LIN {X 0,Y 192.338,Z 600.856,A -85,B 0,C 180,E1 -21672.999,E2 -21672.999} C_VEL
LIN {X 0,Y 190.84,Z 603.624,A -85,B 0,C 180,E1 -21677.23,E2 -21677.23} C_VEL
LIN {X 0,Y 190.204,Z 605.507,A -85,B 0,C 180,E1 -21681.496,E2 -21681.496} C_VEL
LIN {X 0,Y 190.131,Z 606.399,A -85,B 0,C 180,E1 -21686.387,E2 -21686.387} C_VEL
LIN {X 0,Y 190.279,Z 606.289,A -85,B 0,C 180,E1 -21689.995,E2 -21689.995} C_VEL
LIN {X 0,Y 190.157,Z 605.135,A -85,B 0,C 180,E1 -21694.234,E2 -21694.234} C_VEL
LIN {X 0,Y 190.204,Z 603.041,A -85,B 0,C 180,E1 -21698.494,E2 -21698.494} C_VEL
LIN {X 0,Y 191.11,Z 598.889,A -85,B 0,C 180,E1 -21703.824,E2 -21703.824} C_VEL
LIN {X 0,Y 192.967,Z 593.418,A -85,B 0,C 180,E1 -21708.752,E2 -21708.752} C_VEL
LIN {X 0,Y 195.608,Z 586.818,A -85,B 0,C 180,E1 -21713.273,E2 -21713.273} C_VEL
LIN {X 0,Y 198.974,Z 579.355,A -85,B 0,C 180,E1 -21717.327,E2 -21717.327} C_VEL
LIN {X 0,Y 203.185,Z 570.393,A -85,B 0,C 180,E1 -21721.247,E2 -21721.247} C_VEL
LIN {X 0,Y 208.329,Z 559.675,A -85,B 0,C 180,E1 -21724.987,E2 -21724.987} C_VEL
LIN {X 0,Y 213.359,Z 548.57,A -85,B 0,C 180,E1 -21728.117,E2 -21728.117} C_VEL
LIN {X 0,Y 218.295,Z 537.347,A -85,B 0,C 180,E1 -21730.681,E2 -21730.681} C_VEL
LIN {X 0,Y 223.179,Z 525.568,A -85,B 0,C 180,E1 -21732.912,E2 -21732.912} C_VEL
LIN {X 0,Y 228.319,Z 511.73,A -85,B 0,C 180,E1 -21735.062,E2 -21735.062} C_VEL
LIN {X 0,Y 232.885,Z 498.249,A -85,B 0,C 180,E1 -21736.714,E2 -21736.714} C_VEL
LIN {X 0,Y 237.192,Z 482.977,A -85,B 0,C 180,E1 -21738.263,E2 -21738.263} C_VEL
LIN {X 0,Y 240.955,Z 467.509,A -85,B 0,C 180,E1 -21739.471,E2 -21739.471} C_VEL
LIN {X 0,Y 244.029,Z 452.031,A -85,B 0,C 180,E1 -21740.381,E2 -21740.381} C_VEL
LIN {X 0,Y 246.497,Z 435.145,A -85,B 0,C 180,E1 -21741.081,E2 -21741.081} C_VEL
LIN {X 0,Y 248.633,Z 408.344,A -85,B 0,C 180,E1 -21741.862,E2 -21741.862} C_VEL
LIN {X 0,Y 254.712,Z 326.364,A -85,B 0,C 180,E1 -21744.01,E2 -21744.01} C_VEL
LIN {X 0,Y 248.961,Z 314.039,A -85,B 0,C 180,E1 -21746.095,E2 -21746.095} C_VEL
LIN {X 0,Y 242.342,Z 300.931,A -85,B 0,C 180,E1 -21748.648,E2 -21748.648} C_VEL
LIN {X 0,Y 235.672,Z 288.954,A -85,B 0,C 180,E1 -21751.426,E2 -21751.426} C_VEL
LIN {X 0,Y 228.6,Z 278.635,A -85,B 0,C 180,E1 -21754.61,E2 -21754.61} C_VEL
LIN {X 0,Y 222.404,Z 270.045,A -85,B 0,C 180,E1 -21757.717,E2 -21757.717} C_VEL
LIN {X 0,Y 219.05,Z 265.704,A -85,B 0,C 180,E1 -21759.565,E2 -21759.565} C_VEL
LIN {X 0,Y 215.469,Z 261.011,A -85,B 0,C 180,E1 -21761.713,E2 -21761.713} C_VEL
LIN {X 0,Y 212.489,Z 257.254,A -85,B 0,C 180,E1 -21763.628,E2 -21763.628} C_VEL
LIN {X 0,Y 211.602,Z 256.115,A -85,B 0,C 180,E1 -21764.234,E2 -21764.234} C_VEL
LIN {X 0,Y 208.717,Z 252.845,A -85,B 0,C 180,E1 -21766.306,E2 -21766.306} C_VEL
LIN {X 0,Y 207.751,Z 251.108,A -85,B 0,C 180,E1 -21767.113,E2 -21767.113} C_VEL
LIN {X 0,Y 205.027,Z 248.816,A -85,B 0,C 180,E1 -21769.259,E2 -21769.259} C_VEL
LIN {X 0,Y 203.066,Z 245.468,A -85,B 0,C 180,E1 -21771.141,E2 -21771.141} C_VEL
LIN {X 0,Y 200.1,Z 243.192,A -85,B 0,C 180,E1 -21774.079,E2 -21774.079} C_VEL
LIN {X 0,Y 198.632,Z 240.546,A -85,B 0,C 180,E1 -21775.943,E2 -21775.943} C_VEL
LIN {X 0,Y 198.28,Z 239.691,A -85,B 0,C 180,E1 -21776.445,E2 -21776.445} C_VEL
LIN {X 0,Y 194.363,Z 236.846,A -85,B 0,C 180,E1 -21782.332,E2 -21782.332} C_VEL
LIN {X 0,Y 193.15,Z 234.837,A -85,B 0,C 180,E1 -21785.22,E2 -21785.22} C_VEL
LIN {X 0,Y 192.961,Z 233.734,A -85,B 0,C 180,E1 -21786.274,E2 -21786.274} C_VEL
LIN {X 0,Y 192.923,Z 233.731,A -85,B 0,C 180,E1 -21790.436,E2 -21790.436} C_VEL
LIN {X 0,Y 192.737,Z 233.782,A -85,B 0,C 180,E1 -21794.789,E2 -21794.789} C_VEL
LIN {X 0,Y 192.673,Z 233.757,A -85,B 0,C 180,E1 -21799.166,E2 -21799.166} C_VEL
LIN {X 0,Y 192.678,Z 233.917,A -85,B 0,C 180,E1 -21800.694,E2 -21800.694} C_VEL
LIN {X 0,Y 193.05,Z 235.449,A -85,B 0,C 180,E1 -21802.193,E2 -21802.193} C_VEL
LIN {X 0,Y 195.264,Z 238.475,A -85,B 0,C 180,E1 -21807.028,E2 -21807.028} C_VEL
LIN {X 0,Y 198.159,Z 240.092,A -85,B 0,C 180,E1 -21811.032,E2 -21811.032} C_VEL
LIN {X 0,Y 199.513,Z 243.011,A -85,B 0,C 180,E1 -21812.871,E2 -21812.871} C_VEL
LIN {X 0,Y 201.859,Z 245.123,A -85,B 0,C 180,E1 -21815.316,E2 -21815.316} C_VEL
LIN {X 0,Y 203.127,Z 245.924,A -85,B 0,C 180,E1 -21816.49,E2 -21816.49} C_VEL
LIN {X 0,Y 204.819,Z 248.944,A -85,B 0,C 180,E1 -21818.145,E2 -21818.145} C_VEL
LIN {X 0,Y 207.8,Z 251.559,A -85,B 0,C 180,E1 -21820.49,E2 -21820.49} C_VEL
LIN {X 0,Y 209.928,Z 254.781,A -85,B 0,C 180,E1 -21822.166,E2 -21822.166} C_VEL
LIN {X 0,Y 212.127,Z 256.95,A -85,B 0,C 180,E1 -21823.667,E2 -21823.667} C_VEL
LIN {X 0,Y 214.992,Z 260.743,A -85,B 0,C 180,E1 -21825.544,E2 -21825.544} C_VEL
LIN {X 0,Y 216.331,Z 262.284,A -85,B 0,C 180,E1 -21826.367,E2 -21826.367} C_VEL
LIN {X 0,Y 219.522,Z 266.236,A -85,B 0,C 180,E1 -21828.228,E2 -21828.228} C_VEL
LIN {X 0,Y 224.927,Z 273.572,A -85,B 0,C 180,E1 -21831.125,E2 -21831.125} C_VEL
LIN {X 0,Y 232.294,Z 283.876,A -85,B 0,C 180,E1 -21834.615,E2 -21834.615} C_VEL
LIN {X 0,Y 240.584,Z 296.528,A -85,B 0,C 180,E1 -21838.098,E2 -21838.098} C_VEL
LIN {X 0,Y 249.05,Z 310.72,A -85,B 0,C 180,E1 -21841.294,E2 -21841.294} C_VEL
LIN {X 0,Y 254.773,Z 321.054,A -85,B 0,C 180,E1 -21843.283,E2 -21843.283} C_VEL
LIN {X 0,Y 247.206,Z 422.444,A -85,B 0,C 180,E1 -21845.995,E2 -21845.995} C_VEL
LIN {X 0,Y 244.868,Z 439.952,A -85,B 0,C 180,E1 -21846.727,E2 -21846.727} C_VEL
LIN {X 0,Y 241.906,Z 456.256,A -85,B 0,C 180,E1 -21847.712,E2 -21847.712} C_VEL
LIN {X 0,Y 238.609,Z 470.764,A -85,B 0,C 180,E1 -21848.855,E2 -21848.855} C_VEL
LIN {X 0,Y 234.643,Z 485.489,A -85,B 0,C 180,E1 -21850.313,E2 -21850.313} C_VEL
LIN {X 0,Y 229.8,Z 500.689,A -85,B 0,C 180,E1 -21852.197,E2 -21852.197} C_VEL
LIN {X 0,Y 224.715,Z 514.596,A -85,B 0,C 180,E1 -21854.356,E2 -21854.356} C_VEL
LIN {X 0,Y 219.531,Z 527.45,A -85,B 0,C 180,E1 -21856.82,E2 -21856.82} C_VEL
LIN {X 0,Y 214.384,Z 539.21,A -85,B 0,C 180,E1 -21859.573,E2 -21859.573} C_VEL
LIN {X 0,Y 209.27,Z 550.323,A -85,B 0,C 180,E1 -21862.77,E2 -21862.77} C_VEL
LIN {X 0,Y 204.185,Z 560.906,A -85,B 0,C 180,E1 -21866.554,E2 -21866.554} C_VEL
LIN {X 0,Y 199.868,Z 569.725,A -85,B 0,C 180,E1 -21870.509,E2 -21870.509} C_VEL
LIN {X 0,Y 196.827,Z 576.172,A -85,B 0,C 180,E1 -21874.1,E2 -21874.1} C_VEL
LIN {X 0,Y 194.054,Z 582.363,A -85,B 0,C 180,E1 -21878.334,E2 -21878.334} C_VEL
LIN {X 0,Y 192.089,Z 587.269,A -85,B 0,C 180,E1 -21882.686,E2 -21882.686} C_VEL
LIN {X 0,Y 190.687,Z 591.031,A -85,B 0,C 180,E1 -21887.153,E2 -21887.153} C_VEL
LIN {X 0,Y 189.85,Z 593.924,A -85,B 0,C 180,E1 -21892.258,E2 -21892.258} C_VEL
LIN {X 0,Y 189.673,Z 595.396,A -85,B 0,C 180,E1 -21897.215,E2 -21897.215} C_VEL
LIN {X 0,Y 189.927,Z 595.544,A -85,B 0,C 180,E1 -21901.668,E2 -21901.668} C_VEL
LIN {X 0,Y 190.65,Z 594.713,A -85,B 0,C 180,E1 -21906.148,E2 -21906.148} C_VEL
LIN {X 0,Y 192.258,Z 592.527,A -85,B 0,C 180,E1 -21911.152,E2 -21911.152} C_VEL
LIN {X 0,Y 194.891,Z 588.849,A -85,B 0,C 180,E1 -21916.16,E2 -21916.16} C_VEL
LIN {X 0,Y 198.634,Z 583.631,A -85,B 0,C 180,E1 -21921.119,E2 -21921.119} C_VEL
LIN {X 0,Y 202.292,Z 578.64,A -85,B 0,C 180,E1 -21924.735,E2 -21924.735} C_VEL
LIN {X 0,Y 207.752,Z 571.184,A -85,B 0,C 180,E1 -21928.945,E2 -21928.945} C_VEL
LIN {X 0,Y 213.633,Z 562.728,A -85,B 0,C 180,E1 -21932.658,E2 -21932.658} C_VEL
LIN {X 0,Y 219.951,Z 553.243,A -85,B 0,C 180,E1 -21935.967,E2 -21935.967} C_VEL
LIN {X 0,Y 226.201,Z 543.288,A -85,B 0,C 180,E1 -21938.769,E2 -21938.769} C_VEL
LIN {X 0,Y 232.732,Z 531.991,A -85,B 0,C 180,E1 -21941.351,E2 -21941.351} C_VEL
LIN {X 0,Y 239.755,Z 518.558,A -85,B 0,C 180,E1 -21943.802,E2 -21943.802} C_VEL
LIN {X 0,Y 245.931,Z 505.265,A -85,B 0,C 180,E1 -21945.738,E2 -21945.738} C_VEL
LIN {X 0,Y 251.396,Z 491.922,A -85,B 0,C 180,E1 -21947.316,E2 -21947.316} C_VEL
LIN {X 0,Y 256.62,Z 477.172,A -85,B 0,C 180,E1 -21948.717,E2 -21948.717} C_VEL
LIN {X 0,Y 261.421,Z 460.645,A -85,B 0,C 180,E1 -21949.947,E2 -21949.947} C_VEL
LIN {X 0,Y 265.403,Z 443.219,A -85,B 0,C 180,E1 -21950.908,E2 -21950.908} C_VEL
LIN {X 0,Y 268.106,Z 426.904,A -85,B 0,C 180,E1 -21951.542,E2 -21951.542} C_VEL
LIN {X 0,Y 270.551,Z 403.163,A -85,B 0,C 180,E1 -21952.188,E2 -21952.188} C_VEL
LIN {X 0,Y 277.034,Z 332.996,A -85,B 0,C 180,E1 -21953.929,E2 -21953.929} C_VEL
LIN {X 0,Y 273.475,Z 325.887,A -85,B 0,C 180,E1 -21956.161,E2 -21956.161} C_VEL
LIN {X 0,Y 269.912,Z 319.082,A -85,B 0,C 180,E1 -21958.763,E2 -21958.763} C_VEL
LIN {X 0,Y 267.005,Z 313.957,A -85,B 0,C 180,E1 -21961.306,E2 -21961.306} C_VEL
LIN {X 0,Y 264.845,Z 310.049,A -85,B 0,C 180,E1 -21963.668,E2 -21963.668} C_VEL
LIN {X 0,Y 262.881,Z 306.547,A -85,B 0,C 180,E1 -21966.552,E2 -21966.552} C_VEL
LIN {X 0,Y 260.974,Z 304.615,A -85,B 0,C 180,E1 -21971.613,E2 -21971.613} C_VEL
LIN {X 0,Y 260.883,Z 304.439,A -85,B 0,C 180,E1 -21974.17,E2 -21974.17} C_VEL
LIN {X 0,Y 262.656,Z 306.82,A -85,B 0,C 180,E1 -21979.806,E2 -21979.806} C_VEL
LIN {X 0,Y 263.192,Z 308.136,A -85,B 0,C 180,E1 -21980.779,E2 -21980.779} C_VEL
LIN {X 0,Y 263.887,Z 310.312,A -85,B 0,C 180,E1 -21981.966,E2 -21981.966} C_VEL
LIN {X 0,Y 264.943,Z 315.603,A -85,B 0,C 180,E1 -21983.769,E2 -21983.769} C_VEL
LIN {X 0,Y 266.517,Z 322.49,A -85,B 0,C 180,E1 -21985.87,E2 -21985.87} C_VEL
LIN {X 0,Y 267.263,Z 324.416,A -85,B 0,C 180,E1 -21986.606,E2 -21986.606} C_VEL
LIN {X 0,Y 270.175,Z 331.194,A -85,B 0,C 180,E1 -21989.086,E2 -21989.086} C_VEL
LIN {X 0,Y 272.98,Z 338.478,A -85,B 0,C 180,E1 -21991.158,E2 -21991.158} C_VEL
LIN {X 0,Y 273.61,Z 340.153,A -85,B 0,C 180,E1 -21991.596,E2 -21991.596} C_VEL
LIN {X 0,Y 264.902,Z 429.948,A -85,B 0,C 180,E1 -21993.824,E2 -21993.824} C_VEL
LIN {X 0,Y 262.136,Z 446.797,A -85,B 0,C 180,E1 -21994.404,E2 -21994.404} C_VEL
LIN {X 0,Y 258.474,Z 462.569,A -85,B 0,C 180,E1 -21995.119,E2 -21995.119} C_VEL
LIN {X 0,Y 254.221,Z 477.42,A -85,B 0,C 180,E1 -21996.035,E2 -21996.035} C_VEL
LIN {X 0,Y 249.204,Z 491.871,A -85,B 0,C 180,E1 -21997.18,E2 -21997.18} C_VEL
LIN {X 0,Y 243.183,Z 506.787,A -85,B 0,C 180,E1 -21998.708,E2 -21998.708} C_VEL
LIN {X 0,Y 236.767,Z 520.62,A -85,B 0,C 180,E1 -22000.477,E2 -22000.477} C_VEL
LIN {X 0,Y 230.13,Z 533.41,A -85,B 0,C 180,E1 -22002.517,E2 -22002.517} C_VEL
LIN {X 0,Y 223.246,Z 545.379,A -85,B 0,C 180,E1 -22004.898,E2 -22004.898} C_VEL
LIN {X 0,Y 216.347,Z 556.328,A -85,B 0,C 180,E1 -22007.615,E2 -22007.615} C_VEL
LIN {X 0,Y 210.048,Z 565.831,A -85,B 0,C 180,E1 -22010.522,E2 -22010.522} C_VEL
LIN {X 0,Y 203.575,Z 575.118,A -85,B 0,C 180,E1 -22014.059,E2 -22014.059} C_VEL
LIN {X 0,Y 197.908,Z 582.862,A -85,B 0,C 180,E1 -22017.809,E2 -22017.809} C_VEL
LIN {X 0,Y 193.237,Z 589.382,A -85,B 0,C 180,E1 -22021.779,E2 -22021.779} C_VEL
LIN {X 0,Y 189.435,Z 594.752,A -85,B 0,C 180,E1 -22025.91,E2 -22025.91} C_VEL
LIN {X 0,Y 186.424,Z 599.254,A -85,B 0,C 180,E1 -22030.469,E2 -22030.469} C_VEL
LIN {X 0,Y 184.58,Z 602.29,A -85,B 0,C 180,E1 -22034.537,E2 -22034.537} C_VEL
LIN {X 0,Y 183.405,Z 604.538,A -85,B 0,C 180,E1 -22038.949,E2 -22038.949} C_VEL
LIN {X 0,Y 182.996,Z 605.874,A -85,B 0,C 180,E1 -22043.379,E2 -22043.379} C_VEL
LIN {X 0,Y 183.062,Z 606.201,A -85,B 0,C 180,E1 -22047.795,E2 -22047.795} C_VEL
LIN {X 0,Y 183.183,Z 606.04,A -85,B 0,C 180,E1 -22049.995,E2 -22049.995} C_VEL
LIN {X 0,Y 183.068,Z 604.853,A -85,B 0,C 180,E1 -22054.398,E2 -22054.398} C_VEL
LIN {X 0,Y 183.142,Z 602.697,A -85,B 0,C 180,E1 -22058.824,E2 -22058.824} C_VEL
LIN {X 0,Y 183.819,Z 599.432,A -85,B 0,C 180,E1 -22063.256,E2 -22063.256} C_VEL
LIN {X 0,Y 185.369,Z 595.084,A -85,B 0,C 180,E1 -22067.65,E2 -22067.65} C_VEL
LIN {X 0,Y 187.541,Z 589.563,A -85,B 0,C 180,E1 -22072.002,E2 -22072.002} C_VEL
LIN {X 0,Y 190.663,Z 582.691,A -85,B 0,C 180,E1 -22076.246,E2 -22076.246} C_VEL
LIN {X 0,Y 194.678,Z 574.42,A -85,B 0,C 180,E1 -22080.351,E2 -22080.351} C_VEL
LIN {X 0,Y 198.929,Z 565.894,A -85,B 0,C 180,E1 -22083.802,E2 -22083.802} C_VEL
LIN {X 0,Y 203.868,Z 555.818,A -85,B 0,C 180,E1 -22087.098,E2 -22087.098} C_VEL
LIN {X 0,Y 209.39,Z 544.021,A -85,B 0,C 180,E1 -22090.241,E2 -22090.241} C_VEL
LIN {X 0,Y 215.095,Z 531.134,A -85,B 0,C 180,E1 -22092.997,E2 -22092.997} C_VEL
LIN {X 0,Y 220.436,Z 517.973,A -85,B 0,C 180,E1 -22095.273,E2 -22095.273} C_VEL
LIN {X 0,Y 225.856,Z 503.155,A -85,B 0,C 180,E1 -22097.311,E2 -22097.311} C_VEL
LIN {X 0,Y 230.578,Z 488.017,A -85,B 0,C 180,E1 -22098.962,E2 -22098.962} C_VEL
LIN {X 0,Y 234.624,Z 472.527,A -85,B 0,C 180,E1 -22100.295,E2 -22100.295} C_VEL
LIN {X 0,Y 238.167,Z 456.204,A -85,B 0,C 180,E1 -22101.348,E2 -22101.348} C_VEL
LIN {X 0,Y 240.879,Z 439.93,A -85,B 0,C 180,E1 -22102.107,E2 -22102.107} C_VEL
LIN {X 0,Y 242.6,Z 424.068,A -85,B 0,C 180,E1 -22102.634,E2 -22102.634} C_VEL
LIN {X 0,Y 249.846,Z 329.061,A -85,B 0,C 180,E1 -22105.151,E2 -22105.151} C_VEL
LIN {X 0,Y 244.634,Z 317.811,A -85,B 0,C 180,E1 -22107.12,E2 -22107.12} C_VEL
LIN {X 0,Y 238.672,Z 305.728,A -85,B 0,C 180,E1 -22109.543,E2 -22109.543} C_VEL
LIN {X 0,Y 232.267,Z 294.021,A -85,B 0,C 180,E1 -22112.322,E2 -22112.322} C_VEL
LIN {X 0,Y 225.307,Z 283.81,A -85,B 0,C 180,E1 -22115.582,E2 -22115.582} C_VEL
LIN {X 0,Y 219.534,Z 275.617,A -85,B 0,C 180,E1 -22118.623,E2 -22118.623} C_VEL
LIN {X 0,Y 216.458,Z 271.614,A -85,B 0,C 180,E1 -22120.387,E2 -22120.387} C_VEL
LIN {X 0,Y 213.261,Z 267.302,A -85,B 0,C 180,E1 -22122.381,E2 -22122.381} C_VEL
LIN {X 0,Y 210.206,Z 263.314,A -85,B 0,C 180,E1 -22124.43,E2 -22124.43} C_VEL
LIN {X 0,Y 206.577,Z 258.904,A -85,B 0,C 180,E1 -22127.141,E2 -22127.141} C_VEL
LIN {X 0,Y 205.822,Z 257.669,A -85,B 0,C 180,E1 -22127.789,E2 -22127.789} C_VEL
LIN {X 0,Y 203.087,Z 255.091,A -85,B 0,C 180,E1 -22130.037,E2 -22130.037} C_VEL
LIN {X 0,Y 201.38,Z 252.186,A -85,B 0,C 180,E1 -22131.749,E2 -22131.749} C_VEL
LIN {X 0,Y 198.62,Z 249.867,A -85,B 0,C 180,E1 -22134.608,E2 -22134.608} C_VEL
LIN {X 0,Y 197.09,Z 247.122,A -85,B 0,C 180,E1 -22136.613,E2 -22136.613} C_VEL
LIN {X 0,Y 196.883,Z 246.561,A -85,B 0,C 180,E1 -22136.932,E2 -22136.932} C_VEL
LIN {X 0,Y 192.746,Z 243.209,A -85,B 0,C 180,E1 -22143.66,E2 -22143.66} C_VEL
LIN {X 0,Y 191.884,Z 240.983,A -85,B 0,C 180,E1 -22146.309,E2 -22146.309} C_VEL
LIN {X 0,Y 191.289,Z 240.641,A -85,B 0,C 180,E1 -22148.452,E2 -22148.452} C_VEL
LIN {X 0,Y 190.853,Z 240.593,A -85,B 0,C 180,E1 -22157.134,E2 -22157.134} C_VEL
LIN {X 0,Y 191.573,Z 240.923,A -85,B 0,C 180,E1 -22160.258,E2 -22160.258} C_VEL
LIN {X 0,Y 192.487,Z 243.416,A -85,B 0,C 180,E1 -22163.396,E2 -22163.396} C_VEL
LIN {X 0,Y 194.709,Z 245.84,A -85,B 0,C 180,E1 -22167.693,E2 -22167.693} C_VEL
LIN {X 0,Y 196.709,Z 246.907,A -85,B 0,C 180,E1 -22170.459,E2 -22170.459} C_VEL
LIN {X 0,Y 198.309,Z 250.076,A -85,B 0,C 180,E1 -22172.663,E2 -22172.663} C_VEL
LIN {X 0,Y 200.792,Z 252.166,A -85,B 0,C 180,E1 -22175.254,E2 -22175.254} C_VEL
LIN {X 0,Y 201.451,Z 252.625,A -85,B 0,C 180,E1 -22175.886,E2 -22175.886} C_VEL
LIN {X 0,Y 203.509,Z 256.013,A -85,B 0,C 180,E1 -22177.926,E2 -22177.926} C_VEL
LIN {X 0,Y 205.981,Z 258.209,A -85,B 0,C 180,E1 -22179.916,E2 -22179.916} C_VEL
LIN {X 0,Y 208.501,Z 261.797,A -85,B 0,C 180,E1 -22181.921,E2 -22181.921} C_VEL
LIN {X 0,Y 210.143,Z 263.495,A -85,B 0,C 180,E1 -22183.075,E2 -22183.075} C_VEL
LIN {X 0,Y 213.148,Z 267.4,A -85,B 0,C 180,E1 -22185.096,E2 -22185.096} C_VEL
LIN {X 0,Y 217.899,Z 273.568,A -85,B 0,C 180,E1 -22187.991,E2 -22187.991} C_VEL
LIN {X 0,Y 222.398,Z 279.694,A -85,B 0,C 180,E1 -22190.456,E2 -22190.456} C_VEL
LIN {X 0,Y 229.202,Z 289.384,A -85,B 0,C 180,E1 -22193.803,E2 -22193.803} C_VEL
LIN {X 0,Y 236.805,Z 301.176,A -85,B 0,C 180,E1 -22197.142,E2 -22197.142} C_VEL
LIN {X 0,Y 245.252,Z 315.496,A -85,B 0,C 180,E1 -22200.464,E2 -22200.464} C_VEL
LIN {X 0,Y 249.948,Z 324.201,A -85,B 0,C 180,E1 -22202.167,E2 -22202.167} C_VEL
LIN {X 0,Y 242.309,Z 422.38,A -85,B 0,C 180,E1 -22204.792,E2 -22204.792} C_VEL
LIN {X 0,Y 239.966,Z 439.605,A -85,B 0,C 180,E1 -22205.511,E2 -22205.511} C_VEL
LIN {X 0,Y 236.865,Z 456.22,A -85,B 0,C 180,E1 -22206.508,E2 -22206.508} C_VEL
LIN {X 0,Y 233.467,Z 470.849,A -85,B 0,C 180,E1 -22207.669,E2 -22207.669} C_VEL
LIN {X 0,Y 229.364,Z 485.605,A -85,B 0,C 180,E1 -22209.138,E2 -22209.138} C_VEL
LIN {X 0,Y 224.37,Z 500.814,A -85,B 0,C 180,E1 -22211.041,E2 -22211.041} C_VEL
LIN {X 0,Y 219.098,Z 514.743,A -85,B 0,C 180,E1 -22213.226,E2 -22213.226} C_VEL
LIN {X 0,Y 213.737,Z 527.605,A -85,B 0,C 180,E1 -22215.728,E2 -22215.728} C_VEL
LIN {X 0,Y 208.158,Z 539.882,A -85,B 0,C 180,E1 -22218.669,E2 -22218.669} C_VEL
LIN {X 0,Y 203.436,Z 549.794,A -85,B 0,C 180,E1 -22221.562,E2 -22221.562} C_VEL
LIN {X 0,Y 198.084,Z 560.475,A -85,B 0,C 180,E1 -22225.426,E2 -22225.426} C_VEL
LIN {X 0,Y 193.527,Z 569.382,A -85,B 0,C 180,E1 -22229.485,E2 -22229.485} C_VEL
LIN {X 0,Y 190.094,Z 576.283,A -85,B 0,C 180,E1 -22233.399,E2 -22233.399} C_VEL
LIN {X 0,Y 187.323,Z 582.222,A -85,B 0,C 180,E1 -22237.55,E2 -22237.55} C_VEL
LIN {X 0,Y 185.204,Z 587.179,A -85,B 0,C 180,E1 -22242.052,E2 -22242.052} C_VEL
LIN {X 0,Y 183.655,Z 591.194,A -85,B 0,C 180,E1 -22246.921,E2 -22246.921} C_VEL
LIN {X 0,Y 182.953,Z 593.179,A -85,B 0,C 180,E1 -22250.231,E2 -22250.231} C_VEL
LIN {X 0,Y 182.552,Z 595.076,A -85,B 0,C 180,E1 -22255.06,E2 -22255.06} C_VEL
LIN {X 0,Y 182.579,Z 595.63,A -85,B 0,C 180,E1 -22257.705,E2 -22257.705} C_VEL
LIN {X 0,Y 182.905,Z 595.73,A -85,B 0,C 180,E1 -22262.548,E2 -22262.548} C_VEL
LIN {X 0,Y 183.932,Z 594.591,A -85,B 0,C 180,E1 -22267.692,E2 -22267.692} C_VEL
LIN {X 0,Y 185.896,Z 592.13,A -85,B 0,C 180,E1 -22272.888,E2 -22272.888} C_VEL
LIN {X 0,Y 188.963,Z 588.221,A -85,B 0,C 180,E1 -22278.066,E2 -22278.066} C_VEL
LIN {X 0,Y 193.244,Z 582.725,A -85,B 0,C 180,E1 -22283.146,E2 -22283.146} C_VEL
LIN {X 0,Y 197.354,Z 577.429,A -85,B 0,C 180,E1 -22286.816,E2 -22286.816} C_VEL
LIN {X 0,Y 203.36,Z 569.653,A -85,B 0,C 180,E1 -22291.063,E2 -22291.063} C_VEL
LIN {X 0,Y 209.755,Z 560.927,A -85,B 0,C 180,E1 -22294.783,E2 -22294.783} C_VEL
LIN {X 0,Y 216.184,Z 551.655,A -85,B 0,C 180,E1 -22297.904,E2 -22297.904} C_VEL
LIN {X 0,Y 223.192,Z 540.726,A -85,B 0,C 180,E1 -22300.856,E2 -22300.856} C_VEL
LIN {X 0,Y 230.093,Z 528.964,A -85,B 0,C 180,E1 -22303.407,E2 -22303.407} C_VEL
LIN {X 0,Y 236.765,Z 516.49,A -85,B 0,C 180,E1 -22305.571,E2 -22305.571} C_VEL
LIN {X 0,Y 243.028,Z 503.157,A -85,B 0,C 180,E1 -22307.455,E2 -22307.455} C_VEL
LIN {X 0,Y 249.211,Z 488.048,A -85,B 0,C 180,E1 -22309.141,E2 -22309.141} C_VEL
LIN {X 0,Y 254.522,Z 472.824,A -85,B 0,C 180,E1 -22310.463,E2 -22310.463} C_VEL
LIN {X 0,Y 258.895,Z 457.242,A -85,B 0,C 180,E1 -22311.558,E2 -22311.558} C_VEL
LIN {X 0,Y 262.672,Z 440.381,A -85,B 0,C 180,E1 -22312.413,E2 -22312.413} C_VEL
LIN {X 0,Y 265.32,Z 424.212,A -85,B 0,C 180,E1 -22312.991,E2 -22312.991} C_VEL
LIN {X 0,Y 273.799,Z 337.017,A -85,B 0,C 180,E1 -22315.167,E2 -22315.167} C_VEL
LIN {X 0,Y 270.578,Z 330.236,A -85,B 0,C 180,E1 -22317.39,E2 -22317.39} C_VEL
LIN {X 0,Y 267.22,Z 323.674,A -85,B 0,C 180,E1 -22320.122,E2 -22320.122} C_VEL
LIN {X 0,Y 265.134,Z 319.963,A -85,B 0,C 180,E1 -22322.154,E2 -22322.154} C_VEL
LIN {X 0,Y 263.461,Z 316.739,A -85,B 0,C 180,E1 -22324.141,E2 -22324.141} C_VEL
LIN {X 0,Y 261.697,Z 313.482,A -85,B 0,C 180,E1 -22326.883,E2 -22326.883} C_VEL
LIN {X 0,Y 260.013,Z 311.643,A -85,B 0,C 180,E1 -22331.657,E2 -22331.657} C_VEL
LIN {X 0,Y 259.922,Z 311.462,A -85,B 0,C 180,E1 -22334.084,E2 -22334.084} C_VEL
LIN {X 0,Y 261.508,Z 313.724,A -85,B 0,C 180,E1 -22339.501,E2 -22339.501} C_VEL
LIN {X 0,Y 263.884,Z 318.074,A -85,B 0,C 180,E1 -22343.104,E2 -22343.104} C_VEL
LIN {X 0,Y 266.102,Z 322.129,A -85,B 0,C 180,E1 -22345.519,E2 -22345.519} C_VEL
LIN {X 0,Y 267.263,Z 324.416,A -85,B 0,C 180,E1 -22346.606,E2 -22346.606} C_VEL
LIN {X 0,Y 267.892,Z 326.806,A -85,B 0,C 180,E1 -22347.264,E2 -22347.264} C_VEL
LIN {X 0,Y 268.361,Z 332.315,A -85,B 0,C 180,E1 -22348.081,E2 -22348.081} C_VEL
LIN {X 0,Y 268.816,Z 338.044,A -85,B 0,C 180,E1 -22348.867,E2 -22348.867} C_VEL
LIN {X 0,Y 269.495,Z 340.766,A -85,B 0,C 180,E1 -22349.482,E2 -22349.482} C_VEL
LIN {X 0,Y 270.56,Z 343.782,A -85,B 0,C 180,E1 -22350.301,E2 -22350.301} C_VEL
LIN {X 0,Y 261.872,Z 429.959,A -85,B 0,C 180,E1 -22352.427,E2 -22352.427} C_VEL
LIN {X 0,Y 259.007,Z 446.723,A -85,B 0,C 180,E1 -22352.996,E2 -22352.996} C_VEL
LIN {X 0,Y 255.119,Z 462.998,A -85,B 0,C 180,E1 -22353.729,E2 -22353.729} C_VEL
LIN {X 0,Y 250.196,Z 479.349,A -85,B 0,C 180,E1 -22354.748,E2 -22354.748} C_VEL
LIN {X 0,Y 245.067,Z 493.516,A -85,B 0,C 180,E1 -22355.886,E2 -22355.886} C_VEL
LIN {X 0,Y 238.887,Z 508.109,A -85,B 0,C 180,E1 -22357.404,E2 -22357.404} C_VEL
LIN {X 0,Y 232.271,Z 521.623,A -85,B 0,C 180,E1 -22359.159,E2 -22359.159} C_VEL
LIN {X 0,Y 224.804,Z 535.205,A -85,B 0,C 180,E1 -22361.379,E2 -22361.379} C_VEL
LIN {X 0,Y 217.267,Z 547.656,A -85,B 0,C 180,E1 -22363.964,E2 -22363.964} C_VEL
LIN {X 0,Y 210.195,Z 558.331,A -85,B 0,C 180,E1 -22366.726,E2 -22366.726} C_VEL
LIN {X 0,Y 203.741,Z 567.424,A -85,B 0,C 180,E1 -22369.697,E2 -22369.697} C_VEL
LIN {X 0,Y 197.037,Z 576.391,A -85,B 0,C 180,E1 -22373.308,E2 -22373.308} C_VEL
LIN {X 0,Y 190.425,Z 584.967,A -85,B 0,C 180,E1 -22377.766,E2 -22377.766} C_VEL
LIN {X 0,Y 185.845,Z 590.922,A -85,B 0,C 180,E1 -22381.785,E2 -22381.785} C_VEL
LIN {X 0,Y 182.023,Z 595.926,A -85,B 0,C 180,E1 -22386.078,E2 -22386.078} C_VEL
LIN {X 0,Y 178.66,Z 600.732,A -85,B 0,C 180,E1 -22391.652,E2 -22391.652} C_VEL
LIN {X 0,Y 176.873,Z 603.427,A -85,B 0,C 180,E1 -22396.202,E2 -22396.202} C_VEL
LIN {X 0,Y 176.07,Z 605.181,A -85,B 0,C 180,E1 -22400.807,E2 -22400.807} C_VEL
LIN {X 0,Y 175.935,Z 605.954,A -85,B 0,C 180,E1 -22405.412,E2 -22405.412} C_VEL
LIN {X 0,Y 176.089,Z 605.788,A -85,B 0,C 180,E1 -22409.994,E2 -22409.994} C_VEL
LIN {X 0,Y 175.962,Z 604.57,A -85,B 0,C 180,E1 -22414.576,E2 -22414.576} C_VEL
LIN {X 0,Y 176.065,Z 602.348,A -85,B 0,C 180,E1 -22419.182,E2 -22419.182} C_VEL
LIN {X 0,Y 176.85,Z 599.051,A -85,B 0,C 180,E1 -22423.788,E2 -22423.788} C_VEL
LIN {X 0,Y 178.502,Z 594.631,A -85,B 0,C 180,E1 -22428.353,E2 -22428.353} C_VEL
LIN {X 0,Y 180.861,Z 589.067,A -85,B 0,C 180,E1 -22432.86,E2 -22432.86} C_VEL
LIN {X 0,Y 184.199,Z 582.122,A -85,B 0,C 180,E1 -22437.242,E2 -22437.242} C_VEL
LIN {X 0,Y 188.459,Z 573.764,A -85,B 0,C 180,E1 -22441.465,E2 -22441.465} C_VEL
LIN {X 0,Y 193.682,Z 563.771,A -85,B 0,C 180,E1 -22445.484,E2 -22445.484} C_VEL
LIN {X 0,Y 198.982,Z 553.263,A -85,B 0,C 180,E1 -22448.891,E2 -22448.891} C_VEL
LIN {X 0,Y 204.785,Z 541.26,A -85,B 0,C 180,E1 -22451.998,E2 -22451.998} C_VEL
LIN {X 0,Y 209.898,Z 530.05,A -85,B 0,C 180,E1 -22454.335,E2 -22454.335} C_VEL
LIN {X 0,Y 215.521,Z 516.381,A -85,B 0,C 180,E1 -22456.686,E2 -22456.686} C_VEL
LIN {X 0,Y 220.495,Z 503.206,A -85,B 0,C 180,E1 -22458.497,E2 -22458.497} C_VEL
LIN {X 0,Y 225.352,Z 488.099,A -85,B 0,C 180,E1 -22460.163,E2 -22460.163} C_VEL
LIN {X 0,Y 229.51,Z 472.67,A -85,B 0,C 180,E1 -22461.505,E2 -22461.505} C_VEL
LIN {X 0,Y 233.145,Z 456.455,A -85,B 0,C 180,E1 -22462.562,E2 -22462.562} C_VEL
LIN {X 0,Y 235.978,Z 439.989,A -85,B 0,C 180,E1 -22463.337,E2 -22463.337} C_VEL
LIN {X 0,Y 237.821,Z 423.168,A -85,B 0,C 180,E1 -22463.899,E2 -22463.899} C_VEL
LIN {X 0,Y 244.984,Z 331.507,A -85,B 0,C 180,E1 -22466.351,E2 -22466.351} C_VEL
LIN {X 0,Y 237.843,Z 316.115,A -85,B 0,C 180,E1 -22469.256,E2 -22469.256} C_VEL
LIN {X 0,Y 232.102,Z 304.878,A -85,B 0,C 180,E1 -22471.758,E2 -22471.758} C_VEL
LIN {X 0,Y 228.452,Z 298.467,A -85,B 0,C 180,E1 -22473.457,E2 -22473.457} C_VEL
LIN {X 0,Y 220.585,Z 286.664,A -85,B 0,C 180,E1 -22477.384,E2 -22477.384} C_VEL
LIN {X 0,Y 214.909,Z 278.681,A -85,B 0,C 180,E1 -22480.622,E2 -22480.622} C_VEL
LIN {X 0,Y 210.831,Z 273.348,A -85,B 0,C 180,E1 -22483.213,E2 -22483.213} C_VEL
LIN {X 0,Y 207.564,Z 268.996,A -85,B 0,C 180,E1 -22485.531,E2 -22485.531} C_VEL
LIN {X 0,Y 204.587,Z 265.174,A -85,B 0,C 180,E1 -22487.885,E2 -22487.885} C_VEL
LIN {X 0,Y 203.696,Z 264.083,A -85,B 0,C 180,E1 -22488.621,E2 -22488.621} C_VEL
LIN {X 0,Y 201.032,Z 261.119,A -85,B 0,C 180,E1 -22490.981,E2 -22490.981} C_VEL
LIN {X 0,Y 199.762,Z 258.925,A -85,B 0,C 180,E1 -22492.324,E2 -22492.324} C_VEL
LIN {X 0,Y 196.879,Z 256.207,A -85,B 0,C 180,E1 -22495.474,E2 -22495.474} C_VEL
LIN {X 0,Y 195.424,Z 253.388,A -85,B 0,C 180,E1 -22497.522,E2 -22497.522} C_VEL
LIN {X 0,Y 191.442,Z 249.797,A -85,B 0,C 180,E1 -22504.475,E2 -22504.475} C_VEL
LIN {X 0,Y 190.693,Z 247.751,A -85,B 0,C 180,E1 -22507.109,E2 -22507.109} C_VEL
LIN {X 0,Y 189.727,Z 247.592,A -85,B 0,C 180,E1 -22515.638,E2 -22515.638} C_VEL
LIN {X 0,Y 190.519,Z 247.944,A -85,B 0,C 180,E1 -22519.952,E2 -22519.952} C_VEL
LIN {X 0,Y 192.05,Z 251.437,A -85,B 0,C 180,E1 -22524.704,E2 -22524.704} C_VEL
LIN {X 0,Y 195.355,Z 253.866,A -85,B 0,C 180,E1 -22529.993,E2 -22529.993} C_VEL
LIN {X 0,Y 197.129,Z 257.11,A -85,B 0,C 180,E1 -22532.468,E2 -22532.468} C_VEL
LIN {X 0,Y 199.938,Z 259.569,A -85,B 0,C 180,E1 -22535.427,E2 -22535.427} C_VEL
LIN {X 0,Y 202.199,Z 263.022,A -85,B 0,C 180,E1 -22537.695,E2 -22537.695} C_VEL
LIN {X 0,Y 204.228,Z 264.922,A -85,B 0,C 180,E1 -22539.384,E2 -22539.384} C_VEL
LIN {X 0,Y 206.9,Z 268.59,A -85,B 0,C 180,E1 -22541.537,E2 -22541.537} C_VEL
LIN {X 0,Y 208.409,Z 270.348,A -85,B 0,C 180,E1 -22542.643,E2 -22542.643} C_VEL
LIN {X 0,Y 212.425,Z 275.619,A -85,B 0,C 180,E1 -22545.369,E2 -22545.369} C_VEL
LIN {X 0,Y 215.871,Z 280.252,A -85,B 0,C 180,E1 -22547.506,E2 -22547.506} C_VEL
LIN {X 0,Y 219.797,Z 285.639,A -85,B 0,C 180,E1 -22549.722,E2 -22549.722} C_VEL
LIN {X 0,Y 226.449,Z 295.385,A -85,B 0,C 180,E1 -22553.124,E2 -22553.124} C_VEL
LIN {X 0,Y 233.843,Z 307.102,A -85,B 0,C 180,E1 -22556.487,E2 -22556.487} C_VEL
LIN {X 0,Y 241.836,Z 321.008,A -85,B 0,C 180,E1 -22559.743,E2 -22559.743} C_VEL
LIN {X 0,Y 245.131,Z 327.067,A -85,B 0,C 180,E1 -22560.994,E2 -22560.994} C_VEL
LIN {X 0,Y 237.374,Z 423.351,A -85,B 0,C 180,E1 -22563.587,E2 -22563.587} C_VEL
LIN {X 0,Y 234.793,Z 441.379,A -85,B 0,C 180,E1 -22564.358,E2 -22564.358} C_VEL
LIN {X 0,Y 231.586,Z 457.702,A -85,B 0,C 180,E1 -22565.37,E2 -22565.37} C_VEL
LIN {X 0,Y 227.881,Z 472.815,A -85,B 0,C 180,E1 -22566.61,E2 -22566.61} C_VEL
LIN {X 0,Y 223.148,Z 488.836,A -85,B 0,C 180,E1 -22568.286,E2 -22568.286} C_VEL
LIN {X 0,Y 218.529,Z 502.223,A -85,B 0,C 180,E1 -22570.025,E2 -22570.025} C_VEL
LIN {X 0,Y 213.02,Z 516.268,A -85,B 0,C 180,E1 -22572.286,E2 -22572.286} C_VEL
LIN {X 0,Y 207.103,Z 529.746,A -85,B 0,C 180,E1 -22575.009,E2 -22575.009} C_VEL
LIN {X 0,Y 201.608,Z 541.346,A -85,B 0,C 180,E1 -22577.932,E2 -22577.932} C_VEL
LIN {X 0,Y 196.219,Z 552.058,A -85,B 0,C 180,E1 -22581.25,E2 -22581.25} C_VEL
LIN {X 0,Y 191.461,Z 561.159,A -85,B 0,C 180,E1 -22584.694,E2 -22584.694} C_VEL
LIN {X 0,Y 186.689,Z 570.092,A -85,B 0,C 180,E1 -22588.927,E2 -22588.927} C_VEL
LIN {X 0,Y 183.011,Z 577.177,A -85,B 0,C 180,E1 -22593.166,E2 -22593.166} C_VEL
LIN {X 0,Y 179.965,Z 583.402,A -85,B 0,C 180,E1 -22597.861,E2 -22597.861} C_VEL
LIN {X 0,Y 177.873,Z 588.227,A -85,B 0,C 180,E1 -22602.556,E2 -22602.556} C_VEL
LIN {X 0,Y 176.474,Z 591.637,A -85,B 0,C 180,E1 -22607.097,E2 -22607.097} C_VEL
LIN {X 0,Y 175.754,Z 593.85,A -85,B 0,C 180,E1 -22611.098,E2 -22611.098} C_VEL
LIN {X 0,Y 175.431,Z 595.496,A -85,B 0,C 180,E1 -22616.152,E2 -22616.152} C_VEL
LIN {X 0,Y 175.494,Z 595.905,A -85,B 0,C 180,E1 -22618.727,E2 -22618.727} C_VEL
LIN {X 0,Y 176.01,Z 595.85,A -85,B 0,C 180,E1 -22623.993,E2 -22623.993} C_VEL
LIN {X 0,Y 177.327,Z 594.48,A -85,B 0,C 180,E1 -22629.36,E2 -22629.36} C_VEL
LIN {X 0,Y 179.692,Z 591.726,A -85,B 0,C 180,E1 -22634.755,E2 -22634.755} C_VEL
LIN {X 0,Y 183.236,Z 587.503,A -85,B 0,C 180,E1 -22640.1,E2 -22640.1} C_VEL
LIN {X 0,Y 188.096,Z 581.703,A -85,B 0,C 180,E1 -22645.292,E2 -22645.292} C_VEL
LIN {X 0,Y 193.291,Z 575.583,A -85,B 0,C 180,E1 -22649.399,E2 -22649.399} C_VEL
LIN {X 0,Y 199.941,Z 567.263,A -85,B 0,C 180,E1 -22653.687,E2 -22653.687} C_VEL
LIN {X 0,Y 207.52,Z 557.243,A -85,B 0,C 180,E1 -22657.636,E2 -22657.636} C_VEL
LIN {X 0,Y 214.059,Z 547.946,A -85,B 0,C 180,E1 -22660.512,E2 -22660.512} C_VEL
LIN {X 0,Y 221.596,Z 536.308,A -85,B 0,C 180,E1 -22663.414,E2 -22663.414} C_VEL
LIN {X 0,Y 228.64,Z 524.415,A -85,B 0,C 180,E1 -22665.764,E2 -22665.764} C_VEL
LIN {X 0,Y 235.978,Z 510.49,A -85,B 0,C 180,E1 -22667.966,E2 -22667.966} C_VEL
LIN {X 0,Y 242.03,Z 497.24,A -85,B 0,C 180,E1 -22669.636,E2 -22669.636} C_VEL
LIN {X 0,Y 247.695,Z 483.113,A -85,B 0,C 180,E1 -22671.046,E2 -22671.046} C_VEL
LIN {X 0,Y 252.813,Z 467.781,A -85,B 0,C 180,E1 -22672.289,E2 -22672.289} C_VEL
LIN {X 0,Y 256.977,Z 452.622,A -85,B 0,C 180,E1 -22673.229,E2 -22673.229} C_VEL
LIN {X 0,Y 260.396,Z 436.36,A -85,B 0,C 180,E1 -22673.98,E2 -22673.98} C_VEL
LIN {X 0,Y 262.86,Z 419.886,A -85,B 0,C 180,E1 -22674.499,E2 -22674.499} C_VEL
LIN {X 0,Y 270.721,Z 340.881,A -85,B 0,C 180,E1 -22676.466,E2 -22676.466} C_VEL
LIN {X 0,Y 267.151,Z 333.24,A -85,B 0,C 180,E1 -22679.242,E2 -22679.242} C_VEL
LIN {X 0,Y 264.789,Z 328.659,A -85,B 0,C 180,E1 -22681.424,E2 -22681.424} C_VEL
LIN {X 0,Y 262.11,Z 323.4,A -85,B 0,C 180,E1 -22684.613,E2 -22684.613} C_VEL
LIN {X 0,Y 260.594,Z 320.452,A -85,B 0,C 180,E1 -22687.117,E2 -22687.117} C_VEL
LIN {X 0,Y 259.05,Z 318.663,A -85,B 0,C 180,E1 -22691.701,E2 -22691.701} C_VEL
LIN {X 0,Y 258.967,Z 318.526,A -85,B 0,C 180,E1 -22694.137,E2 -22694.137} C_VEL
LIN {X 0,Y 260.404,Z 320.679,A -85,B 0,C 180,E1 -22699.242,E2 -22699.242} C_VEL
LIN {X 0,Y 262.626,Z 324.975,A -85,B 0,C 180,E1 -22702.817,E2 -22702.817} C_VEL
LIN {X 0,Y 264.476,Z 328.431,A -85,B 0,C 180,E1 -22704.919,E2 -22704.919} C_VEL
LIN {X 0,Y 266.208,Z 332.469,A -85,B 0,C 180,E1 -22706.666,E2 -22706.666} C_VEL
LIN {X 0,Y 268.495,Z 338.091,A -85,B 0,C 180,E1 -22708.679,E2 -22708.679} C_VEL
LIN {X 0,Y 269.495,Z 340.766,A -85,B 0,C 180,E1 -22709.482,E2 -22709.482} C_VEL
LIN {X 0,Y 269.778,Z 342.596,A -85,B 0,C 180,E1 -22709.784,E2 -22709.784} C_VEL
LIN {X 0,Y 269.59,Z 345.598,A -85,B 0,C 180,E1 -22709.919,E2 -22709.919} C_VEL
LIN {X 0,Y 268.743,Z 350.082,A -85,B 0,C 180,E1 -22709.812,E2 -22709.812} C_VEL
LIN {X 0,Y 266.624,Z 358.79,A -85,B 0,C 180,E1 -22709.335,E2 -22709.335} C_VEL
LIN {X 0,Y 266.154,Z 361.788,A -85,B 0,C 180,E1 -22709.315,E2 -22709.315} C_VEL
LIN {X 0,Y 258.994,Z 430.583,A -85,B 0,C 180,E1 -22711.009,E2 -22711.009} C_VEL
LIN {X 0,Y 255.999,Z 447.356,A -85,B 0,C 180,E1 -22711.577,E2 -22711.577} C_VEL
LIN {X 0,Y 252.096,Z 463.015,A -85,B 0,C 180,E1 -22712.271,E2 -22712.271} C_VEL
LIN {X 0,Y 246.98,Z 479.458,A -85,B 0,C 180,E1 -22713.288,E2 -22713.288} C_VEL
LIN {X 0,Y 241.055,Z 495.034,A -85,B 0,C 180,E1 -22714.546,E2 -22714.546} C_VEL
LIN {X 0,Y 234.704,Z 509.424,A -85,B 0,C 180,E1 -22716.048,E2 -22716.048} C_VEL
LIN {X 0,Y 227.295,Z 523.849,A -85,B 0,C 180,E1 -22717.954,E2 -22717.954} C_VEL
LIN {X 0,Y 220.213,Z 536.055,A -85,B 0,C 180,E1 -22720.004,E2 -22720.004} C_VEL
LIN {X 0,Y 212.426,Z 548.282,A -85,B 0,C 180,E1 -22722.593,E2 -22722.593} C_VEL
LIN {X 0,Y 205.079,Z 558.826,A -85,B 0,C 180,E1 -22725.365,E2 -22725.365} C_VEL
LIN {X 0,Y 198.352,Z 567.84,A -85,B 0,C 180,E1 -22728.363,E2 -22728.363} C_VEL
LIN {X 0,Y 191.361,Z 576.675,A -85,B 0,C 180,E1 -22732.031,E2 -22732.031} C_VEL
LIN {X 0,Y 185.937,Z 583.277,A -85,B 0,C 180,E1 -22735.456,E2 -22735.456} C_VEL
LIN {X 0,Y 180.666,Z 589.611,A -85,B 0,C 180,E1 -22739.617,E2 -22739.617} C_VEL
LIN {X 0,Y 176.397,Z 594.872,A -85,B 0,C 180,E1 -22744.002,E2 -22744.002} C_VEL
LIN {X 0,Y 172.583,Z 599.698,A -85,B 0,C 180,E1 -22749.488,E2 -22749.488} C_VEL
LIN {X 0,Y 170.787,Z 602.161,A -85,B 0,C 180,E1 -22753.253,E2 -22753.253} C_VEL
LIN {X 0,Y 169.368,Z 604.285,A -85,B 0,C 180,E1 -22758.02,E2 -22758.02} C_VEL
LIN {X 0,Y 168.839,Z 605.547,A -85,B 0,C 180,E1 -22762.821,E2 -22762.821} C_VEL
LIN {X 0,Y 168.884,Z 605.757,A -85,B 0,C 180,E1 -22767.609,E2 -22767.609} C_VEL
LIN {X 0,Y 168.998,Z 605.534,A -85,B 0,C 180,E1 -22769.994,E2 -22769.994} C_VEL
LIN {X 0,Y 168.86,Z 604.284,A -85,B 0,C 180,E1 -22774.769,E2 -22774.769} C_VEL
LIN {X 0,Y 169.012,Z 601.998,A -85,B 0,C 180,E1 -22779.568,E2 -22779.568} C_VEL
LIN {X 0,Y 169.907,Z 598.666,A -85,B 0,C 180,E1 -22784.364,E2 -22784.364} C_VEL
LIN {X 0,Y 171.648,Z 594.169,A -85,B 0,C 180,E1 -22789.114,E2 -22789.114} C_VEL
LIN {X 0,Y 174.214,Z 588.531,A -85,B 0,C 180,E1 -22793.785,E2 -22793.785} C_VEL
LIN {X 0,Y 177.777,Z 581.53,A -85,B 0,C 180,E1 -22798.312,E2 -22798.312} C_VEL
LIN {X 0,Y 182.31,Z 573.073,A -85,B 0,C 180,E1 -22802.655,E2 -22802.655} C_VEL
LIN {X 0,Y 187.847,Z 562.97,A -85,B 0,C 180,E1 -22806.763,E2 -22806.763} C_VEL
LIN {X 0,Y 193.441,Z 552.207,A -85,B 0,C 180,E1 -22810.276,E2 -22810.276} C_VEL
LIN {X 0,Y 199.476,Z 540.234,A -85,B 0,C 180,E1 -22813.387,E2 -22813.387} C_VEL
LIN {X 0,Y 204.813,Z 528.888,A -85,B 0,C 180,E1 -22815.742,E2 -22815.742} C_VEL
LIN {X 0,Y 210.729,Z 514.721,A -85,B 0,C 180,E1 -22818.164,E2 -22818.164} C_VEL
LIN {X 0,Y 216.359,Z 500.01,A -85,B 0,C 180,E1 -22820.112,E2 -22820.112} C_VEL
LIN {X 0,Y 220.757,Z 486.288,A -85,B 0,C 180,E1 -22821.615,E2 -22821.615} C_VEL
LIN {X 0,Y 225.415,Z 469.342,A -85,B 0,C 180,E1 -22823.018,E2 -22823.018} C_VEL
LIN {X 0,Y 228.86,Z 453.653,A -85,B 0,C 180,E1 -22823.979,E2 -22823.979} C_VEL
LIN {X 0,Y 231.616,Z 437.046,A -85,B 0,C 180,E1 -22824.714,E2 -22824.714} C_VEL
LIN {X 0,Y 233.669,Z 415.803,A -85,B 0,C 180,E1 -22825.382,E2 -22825.382} C_VEL
LIN {X 0,Y 240.294,Z 334.389,A -85,B 0,C 180,E1 -22827.555,E2 -22827.555} C_VEL
LIN {X 0,Y 233.598,Z 319.637,A -85,B 0,C 180,E1 -22830.426,E2 -22830.426} C_VEL
LIN {X 0,Y 228.177,Z 308.978,A -85,B 0,C 180,E1 -22832.929,E2 -22832.929} C_VEL
LIN {X 0,Y 225.344,Z 303.917,A -85,B 0,C 180,E1 -22834.302,E2 -22834.302} C_VEL
LIN {X 0,Y 218.014,Z 292.669,A -85,B 0,C 180,E1 -22838.117,E2 -22838.117} C_VEL
LIN {X 0,Y 212.429,Z 284.661,A -85,B 0,C 180,E1 -22841.433,E2 -22841.433} C_VEL
LIN {X 0,Y 208.682,Z 279.626,A -85,B 0,C 180,E1 -22843.906,E2 -22843.906} C_VEL
LIN {X 0,Y 205.383,Z 275.208,A -85,B 0,C 180,E1 -22846.347,E2 -22846.347} C_VEL
LIN {X 0,Y 202.467,Z 271.177,A -85,B 0,C 180,E1 -22848.765,E2 -22848.765} C_VEL
LIN {X 0,Y 199.402,Z 267.753,A -85,B 0,C 180,E1 -22851.552,E2 -22851.552} C_VEL
LIN {X 0,Y 198.356,Z 265.736,A -85,B 0,C 180,E1 -22852.724,E2 -22852.724} C_VEL
LIN {X 0,Y 195.464,Z 262.945,A -85,B 0,C 180,E1 -22855.98,E2 -22855.98} C_VEL
LIN {X 0,Y 193.942,Z 260.181,A -85,B 0,C 180,E1 -22858.184,E2 -22858.184} C_VEL
LIN {X 0,Y 190.156,Z 256.374,A -85,B 0,C 180,E1 -22865.357,E2 -22865.357} C_VEL
LIN {X 0,Y 189.718,Z 254.83,A -85,B 0,C 180,E1 -22867.146,E2 -22867.146} C_VEL
LIN {X 0,Y 188.707,Z 254.62,A -85,B 0,C 180,E1 -22874.491,E2 -22874.491} C_VEL
LIN {X 0,Y 189.469,Z 254.986,A -85,B 0,C 180,E1 -22879.644,E2 -22879.644} C_VEL
LIN {X 0,Y 191.362,Z 258.845,A -85,B 0,C 180,E1 -22885.287,E2 -22885.287} C_VEL
LIN {X 0,Y 194.007,Z 260.742,A -85,B 0,C 180,E1 -22889.499,E2 -22889.499} C_VEL
LIN {X 0,Y 195.85,Z 264.04,A -85,B 0,C 180,E1 -22892.151,E2 -22892.151} C_VEL
LIN {X 0,Y 198.417,Z 266.383,A -85,B 0,C 180,E1 -22894.931,E2 -22894.931} C_VEL
LIN {X 0,Y 200.815,Z 269.924,A -85,B 0,C 180,E1 -22897.388,E2 -22897.388} C_VEL
LIN {X 0,Y 202.424,Z 271.532,A -85,B 0,C 180,E1 -22898.781,E2 -22898.781} C_VEL
LIN {X 0,Y 205.486,Z 275.545,A -85,B 0,C 180,E1 -22901.28,E2 -22901.28} C_VEL
LIN {X 0,Y 210.233,Z 281.913,A -85,B 0,C 180,E1 -22904.695,E2 -22904.695} C_VEL
LIN {X 0,Y 213.761,Z 286.766,A -85,B 0,C 180,E1 -22906.951,E2 -22906.951} C_VEL
LIN {X 0,Y 218.354,Z 293.214,A -85,B 0,C 180,E1 -22909.602,E2 -22909.602} C_VEL
LIN {X 0,Y 224.648,Z 302.915,A -85,B 0,C 180,E1 -22912.894,E2 -22912.894} C_VEL
LIN {X 0,Y 230.868,Z 312.92,A -85,B 0,C 180,E1 -22915.793,E2 -22915.793} C_VEL
LIN {X 0,Y 238.313,Z 326.173,A -85,B 0,C 180,E1 -22918.94,E2 -22918.94} C_VEL
LIN {X 0,Y 240.382,Z 330.371,A -85,B 0,C 180,E1 -22919.784,E2 -22919.784} C_VEL
LIN {X 0,Y 232.703,Z 422.737,A -85,B 0,C 180,E1 -22922.277,E2 -22922.277} C_VEL
LIN {X 0,Y 230.184,Z 440.259,A -85,B 0,C 180,E1 -22923.015,E2 -22923.015} C_VEL
LIN {X 0,Y 227.096,Z 455.894,A -85,B 0,C 180,E1 -22923.955,E2 -22923.955} C_VEL
LIN {X 0,Y 223.468,Z 470.748,A -85,B 0,C 180,E1 -22925.131,E2 -22925.131} C_VEL
LIN {X 0,Y 219.101,Z 485.618,A -85,B 0,C 180,E1 -22926.618,E2 -22926.618} C_VEL
LIN {X 0,Y 213.797,Z 500.874,A -85,B 0,C 180,E1 -22928.555,E2 -22928.555} C_VEL
LIN {X 0,Y 208.033,Z 515.22,A -85,B 0,C 180,E1 -22930.85,E2 -22930.85} C_VEL
LIN {X 0,Y 202.404,Z 527.796,A -85,B 0,C 180,E1 -22933.359,E2 -22933.359} C_VEL
LIN {X 0,Y 196.145,Z 540.604,A -85,B 0,C 180,E1 -22936.538,E2 -22936.538} C_VEL
LIN {X 0,Y 190.502,Z 551.47,A -85,B 0,C 180,E1 -22939.913,E2 -22939.913} C_VEL
LIN {X 0,Y 185.447,Z 560.775,A -85,B 0,C 180,E1 -22943.477,E2 -22943.477} C_VEL
LIN {X 0,Y 180.442,Z 569.713,A -85,B 0,C 180,E1 -22947.773,E2 -22947.773} C_VEL
LIN {X 0,Y 176.41,Z 577.131,A -85,B 0,C 180,E1 -22952.289,E2 -22952.289} C_VEL
LIN {X 0,Y 173.232,Z 583.252,A -85,B 0,C 180,E1 -22956.996,E2 -22956.996} C_VEL
LIN {X 0,Y 170.978,Z 588.128,A -85,B 0,C 180,E1 -22961.865,E2 -22961.865} C_VEL
LIN {X 0,Y 169.312,Z 592.079,A -85,B 0,C 180,E1 -22967.305,E2 -22967.305} C_VEL
LIN {X 0,Y 168.434,Z 594.895,A -85,B 0,C 180,E1 -22973.366,E2 -22973.366} C_VEL
LIN {X 0,Y 168.397,Z 596.093,A -85,B 0,C 180,E1 -22978.783,E2 -22978.783} C_VEL
LIN {X 0,Y 168.844,Z 596.148,A -85,B 0,C 180,E1 -22983.643,E2 -22983.643} C_VEL
LIN {X 0,Y 169.902,Z 595.248,A -85,B 0,C 180,E1 -22988.356,E2 -22988.356} C_VEL
LIN {X 0,Y 172.105,Z 592.988,A -85,B 0,C 180,E1 -22993.969,E2 -22993.969} C_VEL
LIN {X 0,Y 175.542,Z 589.265,A -85,B 0,C 180,E1 -22999.53,E2 -22999.53} C_VEL
LIN {X 0,Y 180.326,Z 583.969,A -85,B 0,C 180,E1 -23004.936,E2 -23004.936} C_VEL
LIN {X 0,Y 184.871,Z 578.906,A -85,B 0,C 180,E1 -23008.805,E2 -23008.805} C_VEL
LIN {X 0,Y 191.479,Z 571.37,A -85,B 0,C 180,E1 -23013.274,E2 -23013.274} C_VEL
LIN {X 0,Y 198.389,Z 562.984,A -85,B 0,C 180,E1 -23017.089,E2 -23017.089} C_VEL
LIN {X 0,Y 204.318,Z 555.309,A -85,B 0,C 180,E1 -23019.88,E2 -23019.88} C_VEL
LIN {X 0,Y 211.561,Z 545.362,A -85,B 0,C 180,E1 -23022.822,E2 -23022.822} C_VEL
LIN {X 0,Y 218.788,Z 534.422,A -85,B 0,C 180,E1 -23025.404,E2 -23025.404} C_VEL
LIN {X 0,Y 226.117,Z 522.19,A -85,B 0,C 180,E1 -23027.72,E2 -23027.72} C_VEL
LIN {X 0,Y 233.111,Z 509.133,A -85,B 0,C 180,E1 -23029.691,E2 -23029.691} C_VEL
LIN {X 0,Y 239,Z 496.558,A -85,B 0,C 180,E1 -23031.232,E2 -23031.232} C_VEL
LIN {X 0,Y 244.925,Z 482.015,A -85,B 0,C 180,E1 -23032.65,E2 -23032.65} C_VEL
LIN {X 0,Y 250.036,Z 467.063,A -85,B 0,C 180,E1 -23033.811,E2 -23033.811} C_VEL
LIN {X 0,Y 254.106,Z 452.614,A -85,B 0,C 180,E1 -23034.689,E2 -23034.689} C_VEL
LIN {X 0,Y 257.566,Z 436.456,A -85,B 0,C 180,E1 -23035.427,E2 -23035.427} C_VEL
LIN {X 0,Y 260.07,Z 420.099,A -85,B 0,C 180,E1 -23035.931,E2 -23035.931} C_VEL
LIN {X 0,Y 267.764,Z 344.927,A -85,B 0,C 180,E1 -23037.795,E2 -23037.795} C_VEL
LIN {X 0,Y 264.301,Z 337.264,A -85,B 0,C 180,E1 -23040.848,E2 -23040.848} C_VEL
LIN {X 0,Y 262.072,Z 332.88,A -85,B 0,C 180,E1 -23043.278,E2 -23043.278} C_VEL
LIN {X 0,Y 260.783,Z 330.118,A -85,B 0,C 180,E1 -23045.074,E2 -23045.074} C_VEL
LIN {X 0,Y 259.441,Z 327.353,A -85,B 0,C 180,E1 -23047.466,E2 -23047.466} C_VEL
LIN {X 0,Y 258.131,Z 325.746,A -85,B 0,C 180,E1 -23051.426,E2 -23051.426} C_VEL
LIN {X 0,Y 258.011,Z 325.448,A -85,B 0,C 180,E1 -23052.586,E2 -23052.586} C_VEL
LIN {X 0,Y 258.105,Z 325.921,A -85,B 0,C 180,E1 -23055.193,E2 -23055.193} C_VEL
LIN {X 0,Y 259.302,Z 327.614,A -85,B 0,C 180,E1 -23058.979,E2 -23058.979} C_VEL
LIN {X 0,Y 261.233,Z 331.553,A -85,B 0,C 180,E1 -23062.3,E2 -23062.3} C_VEL
LIN {X 0,Y 263.282,Z 335.69,A -85,B 0,C 180,E1 -23064.772,E2 -23064.772} C_VEL
LIN {X 0,Y 265.663,Z 341.733,A -85,B 0,C 180,E1 -23067.194,E2 -23067.194} C_VEL
LIN {X 0,Y 267.627,Z 347.368,A -85,B 0,C 180,E1 -23068.962,E2 -23068.962} C_VEL
LIN {X 0,Y 266.154,Z 361.788,A -85,B 0,C 180,E1 -23069.315,E2 -23069.315} C_VEL
LIN {X 0,Y 265.287,Z 367.635,A -85,B 0,C 180,E1 -23069.299,E2 -23069.299} C_VEL
LIN {X 0,Y 261.384,Z 386.794,A -85,B 0,C 180,E1 -23068.601,E2 -23068.601} C_VEL
LIN {X 0,Y 260.52,Z 392.64,A -85,B 0,C 180,E1 -23068.586,E2 -23068.586} C_VEL
LIN {X 0,Y 256.261,Z 431.224,A -85,B 0,C 180,E1 -23069.564,E2 -23069.564} C_VEL
LIN {X 0,Y 253.056,Z 448.438,A -85,B 0,C 180,E1 -23070.14,E2 -23070.14} C_VEL
LIN {X 0,Y 248.731,Z 464.939,A -85,B 0,C 180,E1 -23070.878,E2 -23070.878} C_VEL
LIN {X 0,Y 243.924,Z 479.692,A -85,B 0,C 180,E1 -23071.789,E2 -23071.789} C_VEL
LIN {X 0,Y 237.846,Z 495.182,A -85,B 0,C 180,E1 -23073.02,E2 -23073.02} C_VEL
LIN {X 0,Y 231.308,Z 509.464,A -85,B 0,C 180,E1 -23074.493,E2 -23074.493} C_VEL
LIN {X 0,Y 223.69,Z 523.798,A -85,B 0,C 180,E1 -23076.376,E2 -23076.376} C_VEL
LIN {X 0,Y 215.75,Z 536.924,A -85,B 0,C 180,E1 -23078.571,E2 -23078.571} C_VEL
LIN {X 0,Y 207.715,Z 548.975,A -85,B 0,C 180,E1 -23081.16,E2 -23081.16} C_VEL
LIN {X 0,Y 200.083,Z 559.345,A -85,B 0,C 180,E1 -23083.935,E2 -23083.935} C_VEL
LIN {X 0,Y 192.077,Z 569.562,A -85,B 0,C 180,E1 -23087.453,E2 -23087.453} C_VEL
LIN {X 0,Y 184.917,Z 577.984,A -85,B 0,C 180,E1 -23091.158,E2 -23091.158} C_VEL
LIN {X 0,Y 178.612,Z 585.165,A -85,B 0,C 180,E1 -23095.207,E2 -23095.207} C_VEL
LIN {X 0,Y 173.287,Z 591.171,A -85,B 0,C 180,E1 -23099.533,E2 -23099.533} C_VEL
LIN {X 0,Y 168.048,Z 597.083,A -85,B 0,C 180,E1 -23105.273,E2 -23105.273} C_VEL
LIN {X 0,Y 165.072,Z 600.635,A -85,B 0,C 180,E1 -23110.081,E2 -23110.081} C_VEL
LIN {X 0,Y 163.001,Z 603.252,A -85,B 0,C 180,E1 -23115.002,E2 -23115.002} C_VEL
LIN {X 0,Y 161.956,Z 604.865,A -85,B 0,C 180,E1 -23119.998,E2 -23119.998} C_VEL
LIN {X 0,Y 161.733,Z 605.573,A -85,B 0,C 180,E1 -23125.008,E2 -23125.008} C_VEL
LIN {X 0,Y 161.908,Z 605.276,A -85,B 0,C 180,E1 -23129.994,E2 -23129.994} C_VEL
LIN {X 0,Y 161.808,Z 604.746,A -85,B 0,C 180,E1 -23132.609,E2 -23132.609} C_VEL
LIN {X 0,Y 161.802,Z 602.933,A -85,B 0,C 180,E1 -23137.481,E2 -23137.481} C_VEL
LIN {X 0,Y 162.333,Z 600.089,A -85,B 0,C 180,E1 -23142.495,E2 -23142.495} C_VEL
LIN {X 0,Y 163.796,Z 596.112,A -85,B 0,C 180,E1 -23147.472,E2 -23147.472} C_VEL
LIN {X 0,Y 166.092,Z 590.974,A -85,B 0,C 180,E1 -23152.378,E2 -23152.378} C_VEL
LIN {X 0,Y 169.396,Z 584.636,A -85,B 0,C 180,E1 -23157.146,E2 -23157.146} C_VEL
LIN {X 0,Y 173.982,Z 576.367,A -85,B 0,C 180,E1 -23161.975,E2 -23161.975} C_VEL
LIN {X 0,Y 179.036,Z 567.484,A -85,B 0,C 180,E1 -23166.065,E2 -23166.065} C_VEL
LIN {X 0,Y 184.453,Z 557.836,A -85,B 0,C 180,E1 -23169.649,E2 -23169.649} C_VEL
LIN {X 0,Y 190.501,Z 546.539,A -85,B 0,C 180,E1 -23173.031,E2 -23173.031} C_VEL
LIN {X 0,Y 197.205,Z 533.149,A -85,B 0,C 180,E1 -23176.183,E2 -23176.183} C_VEL
LIN {X 0,Y 203.434,Z 519.495,A -85,B 0,C 180,E1 -23178.701,E2 -23178.701} C_VEL
LIN {X 0,Y 208.888,Z 506.016,A -85,B 0,C 180,E1 -23180.689,E2 -23180.689} C_VEL
LIN {X 0,Y 214.043,Z 491.667,A -85,B 0,C 180,E1 -23182.375,E2 -23182.375} C_VEL
LIN {X 0,Y 218.737,Z 476.188,A -85,B 0,C 180,E1 -23183.819,E2 -23183.819} C_VEL
LIN {X 0,Y 222.666,Z 460.412,A -85,B 0,C 180,E1 -23184.941,E2 -23184.941} C_VEL
LIN {X 0,Y 225.982,Z 443.313,A -85,B 0,C 180,E1 -23185.807,E2 -23185.807} C_VEL
LIN {X 0,Y 228.083,Z 427.17,A -85,B 0,C 180,E1 -23186.389,E2 -23186.389} C_VEL
LIN {X 0,Y 235.635,Z 336.857,A -85,B 0,C 180,E1 -23188.85,E2 -23188.85} C_VEL
LIN {X 0,Y 228.59,Z 321.498,A -85,B 0,C 180,E1 -23192.041,E2 -23192.041} C_VEL
LIN {X 0,Y 222.943,Z 310.394,A -85,B 0,C 180,E1 -23194.834,E2 -23194.834} C_VEL
LIN {X 0,Y 215.486,Z 298.695,A -85,B 0,C 180,E1 -23198.852,E2 -23198.852} C_VEL
LIN {X 0,Y 210.036,Z 290.712,A -85,B 0,C 180,E1 -23202.223,E2 -23202.223} C_VEL
LIN {X 0,Y 206.595,Z 285.983,A -85,B 0,C 180,E1 -23204.584,E2 -23204.584} C_VEL
LIN {X 0,Y 203.467,Z 281.649,A -85,B 0,C 180,E1 -23207.005,E2 -23207.005} C_VEL
LIN {X 0,Y 200.11,Z 277.162,A -85,B 0,C 180,E1 -23209.887,E2 -23209.887} C_VEL
LIN {X 0,Y 197.542,Z 273.923,A -85,B 0,C 180,E1 -23212.414,E2 -23212.414} C_VEL
LIN {X 0,Y 196.801,Z 272.435,A -85,B 0,C 180,E1 -23213.294,E2 -23213.294} C_VEL
LIN {X 0,Y 193.995,Z 269.594,A -85,B 0,C 180,E1 -23216.572,E2 -23216.572} C_VEL
LIN {X 0,Y 192.781,Z 267.156,A -85,B 0,C 180,E1 -23218.434,E2 -23218.434} C_VEL
LIN {X 0,Y 188.978,Z 263.057,A -85,B 0,C 180,E1 -23226.035,E2 -23226.035} C_VEL
LIN {X 0,Y 188.649,Z 261.83,A -85,B 0,C 180,E1 -23227.532,E2 -23227.532} C_VEL
LIN {X 0,Y 187.73,Z 261.628,A -85,B 0,C 180,E1 -23233.288,E2 -23233.288} C_VEL
LIN {X 0,Y 188.421,Z 261.952,A -85,B 0,C 180,E1 -23239.288,E2 -23239.288} C_VEL
LIN {X 0,Y 190.32,Z 265.869,A -85,B 0,C 180,E1 -23245.147,E2 -23245.147} C_VEL
LIN {X 0,Y 192.728,Z 267.731,A -85,B 0,C 180,E1 -23249.108,E2 -23249.108} C_VEL
LIN {X 0,Y 194.571,Z 270.955,A -85,B 0,C 180,E1 -23251.821,E2 -23251.821} C_VEL
LIN {X 0,Y 196.864,Z 273.138,A -85,B 0,C 180,E1 -23254.401,E2 -23254.401} C_VEL
LIN {X 0,Y 199.327,Z 276.721,A -85,B 0,C 180,E1 -23256.977,E2 -23256.977} C_VEL
LIN {X 0,Y 200.704,Z 278.204,A -85,B 0,C 180,E1 -23258.221,E2 -23258.221} C_VEL
LIN {X 0,Y 204.597,Z 283.458,A -85,B 0,C 180,E1 -23261.457,E2 -23261.457} C_VEL
LIN {X 0,Y 208.092,Z 288.258,A -85,B 0,C 180,E1 -23264.024,E2 -23264.024} C_VEL
LIN {X 0,Y 211.662,Z 293.262,A -85,B 0,C 180,E1 -23266.378,E2 -23266.378} C_VEL
LIN {X 0,Y 215.764,Z 299.199,A -85,B 0,C 180,E1 -23268.846,E2 -23268.846} C_VEL
LIN {X 0,Y 221.849,Z 308.754,A -85,B 0,C 180,E1 -23272.148,E2 -23272.148} C_VEL
LIN {X 0,Y 228.297,Z 319.456,A -85,B 0,C 180,E1 -23275.257,E2 -23275.257} C_VEL
LIN {X 0,Y 235.378,Z 332.399,A -85,B 0,C 180,E1 -23278.358,E2 -23278.358} C_VEL
LIN {X 0,Y 235.755,Z 333.111,A -85,B 0,C 180,E1 -23278.513,E2 -23278.513} C_VEL
LIN {X 0,Y 228.007,Z 423.489,A -85,B 0,C 180,E1 -23280.963,E2 -23280.963} C_VEL
LIN {X 0,Y 225.322,Z 441.428,A -85,B 0,C 180,E1 -23281.731,E2 -23281.731} C_VEL
LIN {X 0,Y 222.23,Z 456.453,A -85,B 0,C 180,E1 -23282.651,E2 -23282.651} C_VEL
LIN {X 0,Y 218.092,Z 472.656,A -85,B 0,C 180,E1 -23283.962,E2 -23283.962} C_VEL
LIN {X 0,Y 213.075,Z 488.775,A -85,B 0,C 180,E1 -23285.657,E2 -23285.657} C_VEL
LIN {X 0,Y 208.145,Z 502.25,A -85,B 0,C 180,E1 -23287.42,E2 -23287.42} C_VEL
LIN {X 0,Y 202.35,Z 516.102,A -85,B 0,C 180,E1 -23289.682,E2 -23289.682} C_VEL
LIN {X 0,Y 196.387,Z 528.868,A -85,B 0,C 180,E1 -23292.297,E2 -23292.297} C_VEL
LIN {X 0,Y 190.018,Z 541.4,A -85,B 0,C 180,E1 -23295.507,E2 -23295.507} C_VEL
LIN {X 0,Y 184.111,Z 552.276,A -85,B 0,C 180,E1 -23299.003,E2 -23299.003} C_VEL
LIN {X 0,Y 178.864,Z 561.515,A -85,B 0,C 180,E1 -23302.669,E2 -23302.669} C_VEL
LIN {X 0,Y 173.075,Z 571.391,A -85,B 0,C 180,E1 -23307.678,E2 -23307.678} C_VEL
LIN {X 0,Y 168.85,Z 578.858,A -85,B 0,C 180,E1 -23312.605,E2 -23312.605} C_VEL
LIN {X 0,Y 165.849,Z 584.402,A -85,B 0,C 180,E1 -23317.309,E2 -23317.309} C_VEL
LIN {X 0,Y 163.614,Z 589.082,A -85,B 0,C 180,E1 -23322.408,E2 -23322.408} C_VEL
LIN {X 0,Y 162.106,Z 592.601,A -85,B 0,C 180,E1 -23327.672,E2 -23327.672} C_VEL
LIN {X 0,Y 161.314,Z 595.213,A -85,B 0,C 180,E1 -23333.803,E2 -23333.803} C_VEL
LIN {X 0,Y 161.316,Z 596.323,A -85,B 0,C 180,E1 -23339.384,E2 -23339.384} C_VEL
LIN {X 0,Y 161.857,Z 596.352,A -85,B 0,C 180,E1 -23344.409,E2 -23344.409} C_VEL
LIN {X 0,Y 163.357,Z 595.143,A -85,B 0,C 180,E1 -23350.197,E2 -23350.197} C_VEL
LIN {X 0,Y 166.011,Z 592.604,A -85,B 0,C 180,E1 -23356.035,E2 -23356.035} C_VEL
LIN {X 0,Y 170.009,Z 588.618,A -85,B 0,C 180,E1 -23361.768,E2 -23361.768} C_VEL
LIN {X 0,Y 175.443,Z 583.07,A -85,B 0,C 180,E1 -23367.277,E2 -23367.277} C_VEL
LIN {X 0,Y 180.507,Z 577.782,A -85,B 0,C 180,E1 -23371.175,E2 -23371.175} C_VEL
LIN {X 0,Y 187.705,Z 569.889,A -85,B 0,C 180,E1 -23375.677,E2 -23375.677} C_VEL
LIN {X 0,Y 195.144,Z 561.218,A -85,B 0,C 180,E1 -23379.459,E2 -23379.459} C_VEL
LIN {X 0,Y 202.536,Z 552.02,A -85,B 0,C 180,E1 -23382.611,E2 -23382.611} C_VEL
LIN {X 0,Y 210.463,Z 541.107,A -85,B 0,C 180,E1 -23385.567,E2 -23385.567} C_VEL
LIN {X 0,Y 218.215,Z 529.42,A -85,B 0,C 180,E1 -23388.047,E2 -23388.047} C_VEL
LIN {X 0,Y 225.582,Z 517.009,A -85,B 0,C 180,E1 -23390.168,E2 -23390.168} C_VEL
LIN {X 0,Y 232.668,Z 503.495,A -85,B 0,C 180,E1 -23392.019,E2 -23392.019} C_VEL
LIN {X 0,Y 239.447,Z 488.45,A -85,B 0,C 180,E1 -23393.622,E2 -23393.622} C_VEL
LIN {X 0,Y 245.172,Z 473.322,A -85,B 0,C 180,E1 -23394.883,E2 -23394.883} C_VEL
LIN {X 0,Y 249.709,Z 458.632,A -85,B 0,C 180,E1 -23395.873,E2 -23395.873} C_VEL
LIN {X 0,Y 253.712,Z 442.561,A -85,B 0,C 180,E1 -23396.666,E2 -23396.666} C_VEL
LIN {X 0,Y 256.795,Z 425.682,A -85,B 0,C 180,E1 -23397.254,E2 -23397.254} C_VEL
LIN {X 0,Y 264.237,Z 357.01,A -85,B 0,C 180,E1 -23398.925,E2 -23398.925} C_VEL
LIN {X 0,Y 265.04,Z 349.181,A -85,B 0,C 180,E1 -23399.134,E2 -23399.134} C_VEL
LIN {X 0,Y 262.578,Z 343.418,A -85,B 0,C 180,E1 -23401.533,E2 -23401.533} C_VEL
LIN {X 0,Y 260.445,Z 338.99,A -85,B 0,C 180,E1 -23404.058,E2 -23404.058} C_VEL
LIN {X 0,Y 259.477,Z 336.805,A -85,B 0,C 180,E1 -23405.539,E2 -23405.539} C_VEL
LIN {X 0,Y 258.298,Z 334.244,A -85,B 0,C 180,E1 -23407.818,E2 -23407.818} C_VEL
LIN {X 0,Y 257.099,Z 332.686,A -85,B 0,C 180,E1 -23411.939,E2 -23411.939} C_VEL
LIN {X 0,Y 257.055,Z 332.613,A -85,B 0,C 180,E1 -23414.244,E2 -23414.244} C_VEL
LIN {X 0,Y 258.188,Z 334.509,A -85,B 0,C 180,E1 -23418.669,E2 -23418.669} C_VEL
LIN {X 0,Y 259.972,Z 338.397,A -85,B 0,C 180,E1 -23421.946,E2 -23421.946} C_VEL
LIN {X 0,Y 261.745,Z 342.136,A -85,B 0,C 180,E1 -23424.225,E2 -23424.225} C_VEL
LIN {X 0,Y 264.141,Z 348.735,A -85,B 0,C 180,E1 -23426.834,E2 -23426.834} C_VEL
LIN {X 0,Y 264.939,Z 351.113,A -85,B 0,C 180,E1 -23427.603,E2 -23427.603} C_VEL
LIN {X 0,Y 260.52,Z 392.64,A -85,B 0,C 180,E1 -23428.586,E2 -23428.586} C_VEL
LIN {X 0,Y 259.655,Z 398.503,A -85,B 0,C 180,E1 -23428.561,E2 -23428.561} C_VEL
LIN {X 0,Y 255.783,Z 417.675,A -85,B 0,C 180,E1 -23427.812,E2 -23427.812} C_VEL
LIN {X 0,Y 254.896,Z 423.503,A -85,B 0,C 180,E1 -23427.841,E2 -23427.841} C_VEL
LIN {X 0,Y 252.278,Z 440.344,A -85,B 0,C 180,E1 -23428.329,E2 -23428.329} C_VEL
LIN {X 0,Y 248.49,Z 456.715,A -85,B 0,C 180,E1 -23428.951,E2 -23428.951} C_VEL
LIN {X 0,Y 243.853,Z 472.034,A -85,B 0,C 180,E1 -23429.743,E2 -23429.743} C_VEL
LIN {X 0,Y 238.262,Z 487.191,A -85,B 0,C 180,E1 -23430.78,E2 -23430.78} C_VEL
LIN {X 0,Y 232.124,Z 501.351,A -85,B 0,C 180,E1 -23432.028,E2 -23432.028} C_VEL
LIN {X 0,Y 224.804,Z 515.815,A -85,B 0,C 180,E1 -23433.652,E2 -23433.652} C_VEL
LIN {X 0,Y 217.049,Z 529.092,A -85,B 0,C 180,E1 -23435.552,E2 -23435.552} C_VEL
LIN {X 0,Y 209.041,Z 541.382,A -85,B 0,C 180,E1 -23437.803,E2 -23437.803} C_VEL
LIN {X 0,Y 200.803,Z 552.774,A -85,B 0,C 180,E1 -23440.422,E2 -23440.422} C_VEL
LIN {X 0,Y 192.018,Z 563.879,A -85,B 0,C 180,E1 -23443.704,E2 -23443.704} C_VEL
LIN {X 0,Y 183.103,Z 574.295,A -85,B 0,C 180,E1 -23447.797,E2 -23447.797} C_VEL
LIN {X 0,Y 174.316,Z 583.758,A -85,B 0,C 180,E1 -23452.783,E2 -23452.783} C_VEL
LIN {X 0,Y 168.401,Z 589.902,A -85,B 0,C 180,E1 -23457.138,E2 -23457.138} C_VEL
LIN {X 0,Y 163.562,Z 594.972,A -85,B 0,C 180,E1 -23461.788,E2 -23461.788} C_VEL
LIN {X 0,Y 159.794,Z 598.972,A -85,B 0,C 180,E1 -23466.676,E2 -23466.676} C_VEL
LIN {X 0,Y 157.067,Z 602.002,A -85,B 0,C 180,E1 -23471.741,E2 -23471.741} C_VEL
LIN {X 0,Y 155.35,Z 604.046,A -85,B 0,C 180,E1 -23476.921,E2 -23476.921} C_VEL
LIN {X 0,Y 154.68,Z 605.17,A -85,B 0,C 180,E1 -23482.16,E2 -23482.16} C_VEL
LIN {X 0,Y 154.694,Z 605.31,A -85,B 0,C 180,E1 -23487.39,E2 -23487.39} C_VEL
LIN {X 0,Y 154.809,Z 605.019,A -85,B 0,C 180,E1 -23489.994,E2 -23489.994} C_VEL
LIN {X 0,Y 154.732,Z 604.494,A -85,B 0,C 180,E1 -23492.597,E2 -23492.597} C_VEL
LIN {X 0,Y 154.718,Z 602.605,A -85,B 0,C 180,E1 -23497.826,E2 -23497.826} C_VEL
LIN {X 0,Y 155.333,Z 599.686,A -85,B 0,C 180,E1 -23503.068,E2 -23503.068} C_VEL
LIN {X 0,Y 156.95,Z 595.671,A -85,B 0,C 180,E1 -23508.26,E2 -23508.26} C_VEL
LIN {X 0,Y 159.439,Z 590.451,A -85,B 0,C 180,E1 -23513.366,E2 -23513.366} C_VEL
LIN {X 0,Y 162.99,Z 584.029,A -85,B 0,C 180,E1 -23518.307,E2 -23518.307} C_VEL
LIN {X 0,Y 167.597,Z 576.175,A -85,B 0,C 180,E1 -23523.026,E2 -23523.026} C_VEL
LIN {X 0,Y 173.223,Z 566.716,A -85,B 0,C 180,E1 -23527.478,E2 -23527.478} C_VEL
LIN {X 0,Y 178.932,Z 556.943,A -85,B 0,C 180,E1 -23531.131,E2 -23531.131} C_VEL
LIN {X 0,Y 185.28,Z 545.5,A -85,B 0,C 180,E1 -23534.557,E2 -23534.557} C_VEL
LIN {X 0,Y 191.754,Z 533.021,A -85,B 0,C 180,E1 -23537.518,E2 -23537.518} C_VEL
LIN {X 0,Y 197.629,Z 520.56,A -85,B 0,C 180,E1 -23539.859,E2 -23539.859} C_VEL
LIN {X 0,Y 203.806,Z 505.889,A -85,B 0,C 180,E1 -23542.064,E2 -23542.064} C_VEL
LIN {X 0,Y 209.099,Z 491.539,A -85,B 0,C 180,E1 -23543.76,E2 -23543.76} C_VEL
LIN {X 0,Y 213.923,Z 476.066,A -85,B 0,C 180,E1 -23545.206,E2 -23545.206} C_VEL
LIN {X 0,Y 217.971,Z 460.305,A -85,B 0,C 180,E1 -23546.321,E2 -23546.321} C_VEL
LIN {X 0,Y 221.345,Z 443.357,A -85,B 0,C 180,E1 -23547.181,E2 -23547.181} C_VEL
LIN {X 0,Y 223.528,Z 427.059,A -85,B 0,C 180,E1 -23547.771,E2 -23547.771} C_VEL
LIN {X 0,Y 231.074,Z 339.629,A -85,B 0,C 180,E1 -23550.155,E2 -23550.155} C_VEL
LIN {X 0,Y 224.764,Z 325.586,A -85,B 0,C 180,E1 -23553.196,E2 -23553.196} C_VEL
LIN {X 0,Y 219.714,Z 315.556,A -85,B 0,C 180,E1 -23555.814,E2 -23555.814} C_VEL
LIN {X 0,Y 213.614,Z 305.809,A -85,B 0,C 180,E1 -23559.217,E2 -23559.217} C_VEL
LIN {X 0,Y 209.253,Z 299.109,A -85,B 0,C 180,E1 -23561.965,E2 -23561.965} C_VEL
LIN {X 0,Y 204.491,Z 292.261,A -85,B 0,C 180,E1 -23565.309,E2 -23565.309} C_VEL
LIN {X 0,Y 201.393,Z 287.886,A -85,B 0,C 180,E1 -23567.802,E2 -23567.802} C_VEL
LIN {X 0,Y 198.462,Z 283.802,A -85,B 0,C 180,E1 -23570.439,E2 -23570.439} C_VEL
LIN {X 0,Y 195.868,Z 280.393,A -85,B 0,C 180,E1 -23573.112,E2 -23573.112} C_VEL
LIN {X 0,Y 194.96,Z 278.96,A -85,B 0,C 180,E1 -23574.162,E2 -23574.162} C_VEL
LIN {X 0,Y 192.331,Z 275.884,A -85,B 0,C 180,E1 -23577.486,E2 -23577.486} C_VEL
LIN {X 0,Y 191.273,Z 273.876,A -85,B 0,C 180,E1 -23579.212,E2 -23579.212} C_VEL
LIN {X 0,Y 187.842,Z 269.813,A -85,B 0,C 180,E1 -23586.639,E2 -23586.639} C_VEL
LIN {X 0,Y 187.59,Z 268.83,A -85,B 0,C 180,E1 -23587.923,E2 -23587.923} C_VEL
LIN {X 0,Y 186.831,Z 268.704,A -85,B 0,C 180,E1 -23595.268,E2 -23595.268} C_VEL
LIN {X 0,Y 187.405,Z 269.006,A -85,B 0,C 180,E1 -23599.067,E2 -23599.067} C_VEL
LIN {X 0,Y 189.286,Z 272.901,A -85,B 0,C 180,E1 -23605.019,E2 -23605.019} C_VEL
LIN {X 0,Y 191.415,Z 274.606,A -85,B 0,C 180,E1 -23608.648,E2 -23608.648} C_VEL
LIN {X 0,Y 193.376,Z 277.917,A -85,B 0,C 180,E1 -23611.579,E2 -23611.579} C_VEL
LIN {X 0,Y 195.319,Z 279.866,A -85,B 0,C 180,E1 -23613.851,E2 -23613.851} C_VEL
LIN {X 0,Y 197.816,Z 283.45,A -85,B 0,C 180,E1 -23616.523,E2 -23616.523} C_VEL
LIN {X 0,Y 199.198,Z 285.165,A -85,B 0,C 180,E1 -23617.835,E2 -23617.835} C_VEL
LIN {X 0,Y 202.75,Z 289.993,A -85,B 0,C 180,E1 -23620.863,E2 -23620.863} C_VEL
LIN {X 0,Y 206.119,Z 294.784,A -85,B 0,C 180,E1 -23623.443,E2 -23623.443} C_VEL
LIN {X 0,Y 209.582,Z 299.739,A -85,B 0,C 180,E1 -23625.791,E2 -23625.791} C_VEL
LIN {X 0,Y 213.233,Z 305.195,A -85,B 0,C 180,E1 -23628.085,E2 -23628.085} C_VEL
LIN {X 0,Y 219.779,Z 315.662,A -85,B 0,C 180,E1 -23631.746,E2 -23631.746} C_VEL
LIN {X 0,Y 225.62,Z 325.817,A -85,B 0,C 180,E1 -23634.659,E2 -23634.659} C_VEL
LIN {X 0,Y 231.116,Z 336.059,A -85,B 0,C 180,E1 -23637.18,E2 -23637.18} C_VEL
LIN {X 0,Y 223.502,Z 423.187,A -85,B 0,C 180,E1 -23639.573,E2 -23639.573} C_VEL
LIN {X 0,Y 220.99,Z 439.889,A -85,B 0,C 180,E1 -23640.276,E2 -23640.276} C_VEL
LIN {X 0,Y 217.712,Z 455.775,A -85,B 0,C 180,E1 -23641.218,E2 -23641.218} C_VEL
LIN {X 0,Y 213.384,Z 472.398,A -85,B 0,C 180,E1 -23642.548,E2 -23642.548} C_VEL
LIN {X 0,Y 208.749,Z 487.038,A -85,B 0,C 180,E1 -23644.051,E2 -23644.051} C_VEL
LIN {X 0,Y 203.118,Z 502.172,A -85,B 0,C 180,E1 -23646.018,E2 -23646.018} C_VEL
LIN {X 0,Y 196.806,Z 516.782,A -85,B 0,C 180,E1 -23648.425,E2 -23648.425} C_VEL
LIN {X 0,Y 190.454,Z 529.879,A -85,B 0,C 180,E1 -23651.169,E2 -23651.169} C_VEL
LIN {X 0,Y 184.712,Z 540.743,A -85,B 0,C 180,E1 -23653.993,E2 -23653.993} C_VEL
LIN {X 0,Y 178.595,Z 551.66,A -85,B 0,C 180,E1 -23657.506,E2 -23657.506} C_VEL
LIN {X 0,Y 173.052,Z 561.001,A -85,B 0,C 180,E1 -23661.246,E2 -23661.246} C_VEL
LIN {X 0,Y 167.565,Z 569.976,A -85,B 0,C 180,E1 -23665.797,E2 -23665.797} C_VEL
LIN {X 0,Y 163.569,Z 576.592,A -85,B 0,C 180,E1 -23670.006,E2 -23670.006} C_VEL
LIN {X 0,Y 159.927,Z 582.911,A -85,B 0,C 180,E1 -23675.048,E2 -23675.048} C_VEL
LIN {X 0,Y 157.223,Z 588.02,A -85,B 0,C 180,E1 -23680.44,E2 -23680.44} C_VEL
LIN {X 0,Y 155.434,Z 591.79,A -85,B 0,C 180,E1 -23685.747,E2 -23685.747} C_VEL
LIN {X 0,Y 154.385,Z 594.582,A -85,B 0,C 180,E1 -23691.363,E2 -23691.363} C_VEL
LIN {X 0,Y 154.125,Z 596.173,A -85,B 0,C 180,E1 -23697.135,E2 -23697.135} C_VEL
LIN {X 0,Y 154.266,Z 596.556,A -85,B 0,C 180,E1 -23700.081,E2 -23700.081} C_VEL
LIN {X 0,Y 155.069,Z 596.442,A -85,B 0,C 180,E1 -23706.105,E2 -23706.105} C_VEL
LIN {X 0,Y 156.181,Z 595.648,A -85,B 0,C 180,E1 -23710.092,E2 -23710.092} C_VEL
LIN {X 0,Y 158.37,Z 593.808,A -85,B 0,C 180,E1 -23715.244,E2 -23715.244} C_VEL
LIN {X 0,Y 160.649,Z 591.813,A -85,B 0,C 180,E1 -23718.987,E2 -23718.987} C_VEL
LIN {X 0,Y 166.125,Z 586.706,A -85,B 0,C 180,E1 -23725.567,E2 -23725.567} C_VEL
LIN {X 0,Y 172.067,Z 580.984,A -85,B 0,C 180,E1 -23730.649,E2 -23730.649} C_VEL
LIN {X 0,Y 179.526,Z 573.485,A -85,B 0,C 180,E1 -23735.538,E2 -23735.538} C_VEL
LIN {X 0,Y 187.373,Z 565.047,A -85,B 0,C 180,E1 -23739.678,E2 -23739.678} C_VEL
LIN {X 0,Y 195.723,Z 555.364,A -85,B 0,C 180,E1 -23743.305,E2 -23743.305} C_VEL
LIN {X 0,Y 202.85,Z 546.395,A -85,B 0,C 180,E1 -23745.963,E2 -23745.963} C_VEL
LIN {X 0,Y 211.18,Z 534.813,A -85,B 0,C 180,E1 -23748.691,E2 -23748.691} C_VEL
LIN {X 0,Y 218.843,Z 522.994,A -85,B 0,C 180,E1 -23750.885,E2 -23750.885} C_VEL
LIN {X 0,Y 226.47,Z 509.676,A -85,B 0,C 180,E1 -23752.868,E2 -23752.868} C_VEL
LIN {X 0,Y 233.039,Z 496.567,A -85,B 0,C 180,E1 -23754.412,E2 -23754.412} C_VEL
LIN {X 0,Y 239.591,Z 481.252,A -85,B 0,C 180,E1 -23755.838,E2 -23755.838} C_VEL
LIN {X 0,Y 244.815,Z 466.575,A -85,B 0,C 180,E1 -23756.917,E2 -23756.917} C_VEL
LIN {X 0,Y 248.825,Z 453.093,A -85,B 0,C 180,E1 -23757.69,E2 -23757.69} C_VEL
LIN {X 0,Y 252.345,Z 437.597,A -85,B 0,C 180,E1 -23758.378,E2 -23758.378} C_VEL
LIN {X 0,Y 255.03,Z 421.293,A -85,B 0,C 180,E1 -23758.871,E2 -23758.871} C_VEL
LIN {X 0,Y 262.433,Z 353.502,A -85,B 0,C 180,E1 -23760.52,E2 -23760.52} C_VEL
LIN {X 0,Y 260.548,Z 348.898,A -85,B 0,C 180,E1 -23762.618,E2 -23762.618} C_VEL
LIN {X 0,Y 258.475,Z 343.934,A -85,B 0,C 180,E1 -23765.559,E2 -23765.559} C_VEL
LIN {X 0,Y 257.314,Z 341.294,A -85,B 0,C 180,E1 -23767.848,E2 -23767.848} C_VEL
LIN {X 0,Y 256.101,Z 339.623,A -85,B 0,C 180,E1 -23772.333,E2 -23772.333} C_VEL
LIN {X 0,Y 256.136,Z 339.904,A -85,B 0,C 180,E1 -23774.837,E2 -23774.837} C_VEL
LIN {X 0,Y 257.122,Z 341.516,A -85,B 0,C 180,E1 -23778.466,E2 -23778.466} C_VEL
LIN {X 0,Y 258.75,Z 345.26,A -85,B 0,C 180,E1 -23781.626,E2 -23781.626} C_VEL
LIN {X 0,Y 260.398,Z 349.02,A -85,B 0,C 180,E1 -23783.88,E2 -23783.88} C_VEL
LIN {X 0,Y 262.377,Z 355.057,A -85,B 0,C 180,E1 -23786.223,E2 -23786.223} C_VEL
LIN {X 0,Y 254.896,Z 423.503,A -85,B 0,C 180,E1 -23787.841,E2 -23787.841} C_VEL
LIN {X 0,Y 253.944,Z 429.321,A -85,B 0,C 180,E1 -23787.854,E2 -23787.854} C_VEL
LIN {X 0,Y 249.087,Z 446.309,A -85,B 0,C 180,E1 -23787.233,E2 -23787.233} C_VEL
LIN {X 0,Y 247.395,Z 452.019,A -85,B 0,C 180,E1 -23787.224,E2 -23787.224} C_VEL
LIN {X 0,Y 246.887,Z 453.877,A -85,B 0,C 180,E1 -23787.28,E2 -23787.28} C_VEL
LIN {X 0,Y 242.311,Z 469.347,A -85,B 0,C 180,E1 -23788.013,E2 -23788.013} C_VEL
LIN {X 0,Y 236.923,Z 484.189,A -85,B 0,C 180,E1 -23788.941,E2 -23788.941} C_VEL
LIN {X 0,Y 230.586,Z 498.687,A -85,B 0,C 180,E1 -23790.131,E2 -23790.131} C_VEL
LIN {X 0,Y 223.019,Z 513.465,A -85,B 0,C 180,E1 -23791.691,E2 -23791.691} C_VEL
LIN {X 0,Y 214.993,Z 527.057,A -85,B 0,C 180,E1 -23793.527,E2 -23793.527} C_VEL
LIN {X 0,Y 207.267,Z 538.783,A -85,B 0,C 180,E1 -23795.527,E2 -23795.527} C_VEL
LIN {X 0,Y 198.717,Z 550.451,A -85,B 0,C 180,E1 -23798.097,E2 -23798.097} C_VEL
LIN {X 0,Y 190.523,Z 560.467,A -85,B 0,C 180,E1 -23800.864,E2 -23800.864} C_VEL
LIN {X 0,Y 181.379,Z 570.865,A -85,B 0,C 180,E1 -23804.605,E2 -23804.605} C_VEL
LIN {X 0,Y 174.022,Z 578.663,A -85,B 0,C 180,E1 -23808.207,E2 -23808.207} C_VEL
LIN {X 0,Y 165.436,Z 587.201,A -85,B 0,C 180,E1 -23813.5,E2 -23813.5} C_VEL
LIN {X 0,Y 158.469,Z 593.925,A -85,B 0,C 180,E1 -23819.329,E2 -23819.329} C_VEL
LIN {X 0,Y 153.202,Z 598.994,A -85,B 0,C 180,E1 -23825.609,E2 -23825.609} C_VEL
LIN {X 0,Y 150.259,Z 601.929,A -85,B 0,C 180,E1 -23830.882,E2 -23830.882} C_VEL
LIN {X 0,Y 148.37,Z 603.932,A -85,B 0,C 180,E1 -23836.294,E2 -23836.294} C_VEL
LIN {X 0,Y 147.604,Z 604.98,A -85,B 0,C 180,E1 -23841.781,E2 -23841.781} C_VEL
LIN {X 0,Y 147.604,Z 605.084,A -85,B 0,C 180,E1 -23847.264,E2 -23847.264} C_VEL
LIN {X 0,Y 147.655,Z 604.457,A -85,B 0,C 180,E1 -23851.769,E2 -23851.769} C_VEL
LIN {X 0,Y 147.566,Z 603.393,A -85,B 0,C 180,E1 -23855.459,E2 -23855.459} C_VEL
LIN {X 0,Y 147.883,Z 600.892,A -85,B 0,C 180,E1 -23860.951,E2 -23860.951} C_VEL
LIN {X 0,Y 149.135,Z 597.396,A -85,B 0,C 180,E1 -23866.417,E2 -23866.417} C_VEL
LIN {X 0,Y 151.342,Z 592.701,A -85,B 0,C 180,E1 -23871.801,E2 -23871.801} C_VEL
LIN {X 0,Y 154.616,Z 586.803,A -85,B 0,C 180,E1 -23877.027,E2 -23877.027} C_VEL
LIN {X 0,Y 159.004,Z 579.621,A -85,B 0,C 180,E1 -23882.024,E2 -23882.024} C_VEL
LIN {X 0,Y 164.43,Z 570.894,A -85,B 0,C 180,E1 -23886.745,E2 -23886.745} C_VEL
LIN {X 0,Y 170.074,Z 561.839,A -85,B 0,C 180,E1 -23890.596,E2 -23890.596} C_VEL
LIN {X 0,Y 176.658,Z 550.569,A -85,B 0,C 180,E1 -23894.444,E2 -23894.444} C_VEL
LIN {X 0,Y 183.245,Z 538.842,A -85,B 0,C 180,E1 -23897.576,E2 -23897.576} C_VEL
LIN {X 0,Y 189.739,Z 526.316,A -85,B 0,C 180,E1 -23900.217,E2 -23900.217} C_VEL
LIN {X 0,Y 195.91,Z 512.715,A -85,B 0,C 180,E1 -23902.522,E2 -23902.522} C_VEL
LIN {X 0,Y 201.921,Z 498.089,A -85,B 0,C 180,E1 -23904.436,E2 -23904.436} C_VEL
LIN {X 0,Y 206.737,Z 484.041,A -85,B 0,C 180,E1 -23905.946,E2 -23905.946} C_VEL
LIN {X 0,Y 211.488,Z 467.943,A -85,B 0,C 180,E1 -23907.251,E2 -23907.251} C_VEL
LIN {X 0,Y 215.467,Z 450.829,A -85,B 0,C 180,E1 -23908.269,E2 -23908.269} C_VEL
LIN {X 0,Y 218.355,Z 433.711,A -85,B 0,C 180,E1 -23908.975,E2 -23908.975} C_VEL
LIN {X 0,Y 221.157,Z 404.235,A -85,B 0,C 180,E1 -23909.845,E2 -23909.845} C_VEL
LIN {X 0,Y 226.636,Z 342.548,A -85,B 0,C 180,E1 -23911.506,E2 -23911.506} C_VEL
LIN {X 0,Y 220.869,Z 329.333,A -85,B 0,C 180,E1 -23914.452,E2 -23914.452} C_VEL
LIN {X 0,Y 216.594,Z 320.776,A -85,B 0,C 180,E1 -23916.801,E2 -23916.801} C_VEL
LIN {X 0,Y 210.338,Z 310.487,A -85,B 0,C 180,E1 -23920.481,E2 -23920.481} C_VEL
LIN {X 0,Y 205.648,Z 303.202,A -85,B 0,C 180,E1 -23923.628,E2 -23923.628} C_VEL
LIN {X 0,Y 201.573,Z 297.325,A -85,B 0,C 180,E1 -23926.737,E2 -23926.737} C_VEL
LIN {X 0,Y 199.393,Z 294.136,A -85,B 0,C 180,E1 -23928.579,E2 -23928.579} C_VEL
LIN {X 0,Y 196.724,Z 290.359,A -85,B 0,C 180,E1 -23931.097,E2 -23931.097} C_VEL
LIN {X 0,Y 194.086,Z 286.667,A -85,B 0,C 180,E1 -23933.95,E2 -23933.95} C_VEL
LIN {X 0,Y 193.412,Z 285.652,A -85,B 0,C 180,E1 -23934.766,E2 -23934.766} C_VEL
LIN {X 0,Y 190.831,Z 282.355,A -85,B 0,C 180,E1 -23938.237,E2 -23938.237} C_VEL
LIN {X 0,Y 190.033,Z 280.763,A -85,B 0,C 180,E1 -23939.604,E2 -23939.604} C_VEL
LIN {X 0,Y 186.767,Z 276.69,A -85,B 0,C 180,E1 -23947.065,E2 -23947.065} C_VEL
LIN {X 0,Y 186.613,Z 275.934,A -85,B 0,C 180,E1 -23947.965,E2 -23947.965} C_VEL
LIN {X 0,Y 185.829,Z 275.695,A -85,B 0,C 180,E1 -23953.117,E2 -23953.117} C_VEL
LIN {X 0,Y 186.396,Z 276.034,A -85,B 0,C 180,E1 -23958.844,E2 -23958.844} C_VEL
LIN {X 0,Y 188.254,Z 279.918,A -85,B 0,C 180,E1 -23964.889,E2 -23964.889} C_VEL
LIN {X 0,Y 190.147,Z 281.539,A -85,B 0,C 180,E1 -23968.238,E2 -23968.238} C_VEL
LIN {X 0,Y 192.145,Z 284.854,A -85,B 0,C 180,E1 -23971.286,E2 -23971.286} C_VEL
LIN {X 0,Y 193.88,Z 286.707,A -85,B 0,C 180,E1 -23973.396,E2 -23973.396} C_VEL
LIN {X 0,Y 196.392,Z 290.318,A -85,B 0,C 180,E1 -23976.143,E2 -23976.143} C_VEL
LIN {X 0,Y 197.735,Z 292.17,A -85,B 0,C 180,E1 -23977.476,E2 -23977.476} C_VEL
LIN {X 0,Y 200.808,Z 296.436,A -85,B 0,C 180,E1 -23980.193,E2 -23980.193} C_VEL
LIN {X 0,Y 204.665,Z 302,A -85,B 0,C 180,E1 -23983.216,E2 -23983.216} C_VEL
LIN {X 0,Y 209.805,Z 309.696,A -85,B 0,C 180,E1 -23986.709,E2 -23986.709} C_VEL
LIN {X 0,Y 215.325,Z 318.654,A -85,B 0,C 180,E1 -23990.022,E2 -23990.022} C_VEL
LIN {X 0,Y 221.76,Z 329.848,A -85,B 0,C 180,E1 -23993.453,E2 -23993.453} C_VEL
LIN {X 0,Y 226.733,Z 339.245,A -85,B 0,C 180,E1 -23995.855,E2 -23995.855} C_VEL
LIN {X 0,Y 218.987,Z 424.117,A -85,B 0,C 180,E1 -23998.168,E2 -23998.168} C_VEL
LIN {X 0,Y 216.289,Z 441.123,A -85,B 0,C 180,E1 -23998.885,E2 -23998.885} C_VEL
LIN {X 0,Y 212.745,Z 457.575,A -85,B 0,C 180,E1 -23999.893,E2 -23999.893} C_VEL
LIN {X 0,Y 208.348,Z 473.652,A -85,B 0,C 180,E1 -24001.209,E2 -24001.209} C_VEL
LIN {X 0,Y 203.442,Z 488.474,A -85,B 0,C 180,E1 -24002.766,E2 -24002.766} C_VEL
LIN {X 0,Y 198.213,Z 502.066,A -85,B 0,C 180,E1 -24004.544,E2 -24004.544} C_VEL
LIN {X 0,Y 191.566,Z 516.959,A -85,B 0,C 180,E1 -24007.007,E2 -24007.007} C_VEL
LIN {X 0,Y 185.127,Z 529.845,A -85,B 0,C 180,E1 -24009.738,E2 -24009.738} C_VEL
LIN {X 0,Y 178.673,Z 541.591,A -85,B 0,C 180,E1 -24012.848,E2 -24012.848} C_VEL
LIN {X 0,Y 172.319,Z 552.408,A -85,B 0,C 180,E1 -24016.443,E2 -24016.443} C_VEL
LIN {X 0,Y 166.574,Z 561.696,A -85,B 0,C 180,E1 -24020.29,E2 -24020.29} C_VEL
LIN {X 0,Y 160.863,Z 570.593,A -85,B 0,C 180,E1 -24024.993,E2 -24024.993} C_VEL
LIN {X 0,Y 156.169,Z 577.975,A -85,B 0,C 180,E1 -24030.006,E2 -24030.006} C_VEL
LIN {X 0,Y 152.514,Z 584.046,A -85,B 0,C 180,E1 -24035.294,E2 -24035.294} C_VEL
LIN {X 0,Y 149.908,Z 588.904,A -85,B 0,C 180,E1 -24040.815,E2 -24040.815} C_VEL
LIN {X 0,Y 148.097,Z 592.553,A -85,B 0,C 180,E1 -24046.549,E2 -24046.549} C_VEL
LIN {X 0,Y 147.179,Z 595.128,A -85,B 0,C 180,E1 -24052.464,E2 -24052.464} C_VEL
LIN {X 0,Y 147.027,Z 596.013,A -85,B 0,C 180,E1 -24055.487,E2 -24055.487} C_VEL
LIN {X 0,Y 147.247,Z 596.851,A -85,B 0,C 180,E1 -24061.676,E2 -24061.676} C_VEL
LIN {X 0,Y 148.412,Z 596.478,A -85,B 0,C 180,E1 -24068.003,E2 -24068.003} C_VEL
LIN {X 0,Y 150.73,Z 594.837,A -85,B 0,C 180,E1 -24074.385,E2 -24074.385} C_VEL
LIN {X 0,Y 154.52,Z 591.831,A -85,B 0,C 180,E1 -24080.65,E2 -24080.65} C_VEL
LIN {X 0,Y 159.795,Z 587.301,A -85,B 0,C 180,E1 -24086.691,E2 -24086.691} C_VEL
LIN {X 0,Y 166.7,Z 581.133,A -85,B 0,C 180,E1 -24092.369,E2 -24092.369} C_VEL
LIN {X 0,Y 173.376,Z 574.841,A -85,B 0,C 180,E1 -24096.622,E2 -24096.622} C_VEL
LIN {X 0,Y 180.812,Z 567.438,A -85,B 0,C 180,E1 -24100.498,E2 -24100.498} C_VEL
LIN {X 0,Y 189.757,Z 557.736,A -85,B 0,C 180,E1 -24104.367,E2 -24104.367} C_VEL
LIN {X 0,Y 197.766,Z 548.17,A -85,B 0,C 180,E1 -24107.306,E2 -24107.306} C_VEL
LIN {X 0,Y 206.344,Z 536.919,A -85,B 0,C 180,E1 -24110.03,E2 -24110.03} C_VEL
LIN {X 0,Y 214.523,Z 524.961,A -85,B 0,C 180,E1 -24112.304,E2 -24112.304} C_VEL
LIN {X 0,Y 221.992,Z 512.632,A -85,B 0,C 180,E1 -24114.173,E2 -24114.173} C_VEL
LIN {X 0,Y 228.21,Z 500.97,A -85,B 0,C 180,E1 -24115.607,E2 -24115.607} C_VEL
LIN {X 0,Y 234.56,Z 487.521,A -85,B 0,C 180,E1 -24116.933,E2 -24116.933} C_VEL
LIN {X 0,Y 240.53,Z 472.294,A -85,B 0,C 180,E1 -24118.134,E2 -24118.134} C_VEL
LIN {X 0,Y 245.254,Z 457.553,A -85,B 0,C 180,E1 -24119.038,E2 -24119.038} C_VEL
LIN {X 0,Y 249.502,Z 440.738,A -85,B 0,C 180,E1 -24119.798,E2 -24119.798} C_VEL
LIN {X 0,Y 252.414,Z 425.042,A -85,B 0,C 180,E1 -24120.301,E2 -24120.301} C_VEL
LIN {X 0,Y 260.091,Z 357.929,A -85,B 0,C 180,E1 -24121.908,E2 -24121.908} C_VEL
LIN {X 0,Y 258.106,Z 353.089,A -85,B 0,C 180,E1 -24124.481,E2 -24124.481} C_VEL
LIN {X 0,Y 256.917,Z 350.132,A -85,B 0,C 180,E1 -24126.493,E2 -24126.493} C_VEL
LIN {X 0,Y 256.171,Z 348.161,A -85,B 0,C 180,E1 -24128.233,E2 -24128.233} C_VEL
LIN {X 0,Y 255.118,Z 346.549,A -85,B 0,C 180,E1 -24132.731,E2 -24132.731} C_VEL
LIN {X 0,Y 255.339,Z 347.372,A -85,B 0,C 180,E1 -24135.976,E2 -24135.976} C_VEL
LIN {X 0,Y 256.033,Z 348.414,A -85,B 0,C 180,E1 -24138.176,E2 -24138.176} C_VEL
LIN {X 0,Y 257.483,Z 352.008,A -85,B 0,C 180,E1 -24141.218,E2 -24141.218} C_VEL
LIN {X 0,Y 258.835,Z 355.33,A -85,B 0,C 180,E1 -24143.245,E2 -24143.245} C_VEL
LIN {X 0,Y 260.03,Z 359.122,A -85,B 0,C 180,E1 -24144.802,E2 -24144.802} C_VEL
LIN {X 0,Y 251.94,Z 429.602,A -85,B 0,C 180,E1 -24146.473,E2 -24146.473} C_VEL
LIN {X 0,Y 248.758,Z 446.379,A -85,B 0,C 180,E1 -24147.012,E2 -24147.012} C_VEL
LIN {X 0,Y 246.887,Z 453.877,A -85,B 0,C 180,E1 -24147.28,E2 -24147.28} C_VEL
LIN {X 0,Y 246.118,Z 456.425,A -85,B 0,C 180,E1 -24147.3,E2 -24147.3} C_VEL
LIN {X 0,Y 244.106,Z 461.335,A -85,B 0,C 180,E1 -24147.093,E2 -24147.093} C_VEL
LIN {X 0,Y 240.201,Z 469.66,A -85,B 0,C 180,E1 -24146.565,E2 -24146.565} C_VEL
LIN {X 0,Y 238.734,Z 473.355,A -85,B 0,C 180,E1 -24146.621,E2 -24146.621} C_VEL
LIN {X 0,Y 232.921,Z 487.98,A -85,B 0,C 180,E1 -24147.578,E2 -24147.578} C_VEL
LIN {X 0,Y 226.488,Z 501.869,A -85,B 0,C 180,E1 -24148.759,E2 -24148.759} C_VEL
LIN {X 0,Y 218.749,Z 516.179,A -85,B 0,C 180,E1 -24150.289,E2 -24150.289} C_VEL
LIN {X 0,Y 209.881,Z 530.318,A -85,B 0,C 180,E1 -24152.268,E2 -24152.268} C_VEL
LIN {X 0,Y 201.993,Z 541.423,A -85,B 0,C 180,E1 -24154.27,E2 -24154.27} C_VEL
LIN {X 0,Y 191.954,Z 554.156,A -85,B 0,C 180,E1 -24157.213,E2 -24157.213} C_VEL
LIN {X 0,Y 182.495,Z 564.916,A -85,B 0,C 180,E1 -24160.479,E2 -24160.479} C_VEL
LIN {X 0,Y 174.903,Z 572.959,A -85,B 0,C 180,E1 -24163.668,E2 -24163.668} C_VEL
LIN {X 0,Y 166.827,Z 580.785,A -85,B 0,C 180,E1 -24167.615,E2 -24167.615} C_VEL
LIN {X 0,Y 159.738,Z 587.409,A -85,B 0,C 180,E1 -24171.972,E2 -24171.972} C_VEL
LIN {X 0,Y 152.324,Z 594.037,A -85,B 0,C 180,E1 -24177.948,E2 -24177.948} C_VEL
LIN {X 0,Y 146.689,Z 599.018,A -85,B 0,C 180,E1 -24184.45,E2 -24184.45} C_VEL
LIN {X 0,Y 143.494,Z 601.866,A -85,B 0,C 180,E1 -24189.943,E2 -24189.943} C_VEL
LIN {X 0,Y 141.408,Z 603.825,A -85,B 0,C 180,E1 -24195.605,E2 -24195.605} C_VEL
LIN {X 0,Y 140.528,Z 604.79,A -85,B 0,C 180,E1 -24201.364,E2 -24201.364} C_VEL
LIN {X 0,Y 140.498,Z 604.858,A -85,B 0,C 180,E1 -24207.126,E2 -24207.126} C_VEL
LIN {X 0,Y 140.575,Z 604.345,A -85,B 0,C 180,E1 -24210.928,E2 -24210.928} C_VEL
LIN {X 0,Y 140.487,Z 603.058,A -85,B 0,C 180,E1 -24215.735,E2 -24215.735} C_VEL
LIN {X 0,Y 140.842,Z 600.509,A -85,B 0,C 180,E1 -24221.506,E2 -24221.506} C_VEL
LIN {X 0,Y 142.773,Z 595.838,A -85,B 0,C 180,E1 -24228.653,E2 -24228.653} C_VEL
LIN {X 0,Y 145.444,Z 590.81,A -85,B 0,C 180,E1 -24234.242,E2 -24234.242} C_VEL
LIN {X 0,Y 149.269,Z 584.537,A -85,B 0,C 180,E1 -24239.619,E2 -24239.619} C_VEL
LIN {X 0,Y 154.722,Z 576.094,A -85,B 0,C 180,E1 -24245.155,E2 -24245.155} C_VEL
LIN {X 0,Y 160.282,Z 567.609,A -85,B 0,C 180,E1 -24249.469,E2 -24249.469} C_VEL
LIN {X 0,Y 166.405,Z 558.1,A -85,B 0,C 180,E1 -24253.328,E2 -24253.328} C_VEL
LIN {X 0,Y 173.181,Z 546.91,A -85,B 0,C 180,E1 -24256.915,E2 -24256.915} C_VEL
LIN {X 0,Y 179.489,Z 535.657,A -85,B 0,C 180,E1 -24259.766,E2 -24259.766} C_VEL
LIN {X 0,Y 185.734,Z 523.804,A -85,B 0,C 180,E1 -24262.164,E2 -24262.164} C_VEL
LIN {X 0,Y 192.192,Z 509.884,A -85,B 0,C 180,E1 -24264.44,E2 -24264.44} C_VEL
LIN {X 0,Y 197.76,Z 496.293,A -85,B 0,C 180,E1 -24266.158,E2 -24266.158} C_VEL
LIN {X 0,Y 203.126,Z 480.879,A -85,B 0,C 180,E1 -24267.715,E2 -24267.715} C_VEL
LIN {X 0,Y 207.655,Z 465.162,A -85,B 0,C 180,E1 -24268.934,E2 -24268.934} C_VEL
LIN {X 0,Y 211.349,Z 449.442,A -85,B 0,C 180,E1 -24269.822,E2 -24269.822} C_VEL
LIN {X 0,Y 214.284,Z 431.895,A -85,B 0,C 180,E1 -24270.531,E2 -24270.531} C_VEL
LIN {X 0,Y 222.314,Z 345.44,A -85,B 0,C 180,E1 -24272.903,E2 -24272.903} C_VEL
LIN {X 0,Y 217.094,Z 333.202,A -85,B 0,C 180,E1 -24275.74,E2 -24275.74} C_VEL
LIN {X 0,Y 213.672,Z 326.278,A -85,B 0,C 180,E1 -24277.712,E2 -24277.712} C_VEL
LIN {X 0,Y 207.616,Z 316.064,A -85,B 0,C 180,E1 -24281.468,E2 -24281.468} C_VEL
LIN {X 0,Y 203.203,Z 309.109,A -85,B 0,C 180,E1 -24284.561,E2 -24284.561} C_VEL
LIN {X 0,Y 199.21,Z 303.059,A -85,B 0,C 180,E1 -24287.78,E2 -24287.78} C_VEL
LIN {X 0,Y 195.292,Z 297.155,A -85,B 0,C 180,E1 -24291.494,E2 -24291.494} C_VEL
LIN {X 0,Y 192.559,Z 293.366,A -85,B 0,C 180,E1 -24294.525,E2 -24294.525} C_VEL
LIN {X 0,Y 191.727,Z 292.144,A -85,B 0,C 180,E1 -24295.582,E2 -24295.582} C_VEL
LIN {X 0,Y 189.305,Z 288.738,A -85,B 0,C 180,E1 -24299.081,E2 -24299.081} C_VEL
LIN {X 0,Y 188.651,Z 287.52,A -85,B 0,C 180,E1 -24300.252,E2 -24300.252} C_VEL
LIN {X 0,Y 185.707,Z 283.574,A -85,B 0,C 180,E1 -24307.477,E2 -24307.477} C_VEL
LIN {X 0,Y 185.483,Z 282.794,A -85,B 0,C 180,E1 -24308.719,E2 -24308.719} C_VEL
LIN {X 0,Y 185.355,Z 282.924,A -85,B 0,C 180,E1 -24318.386,E2 -24318.386} C_VEL
LIN {X 0,Y 187.067,Z 286.764,A -85,B 0,C 180,E1 -24324.411,E2 -24324.411} C_VEL
LIN {X 0,Y 188.882,Z 288.394,A -85,B 0,C 180,E1 -24327.796,E2 -24327.796} C_VEL
LIN {X 0,Y 190.837,Z 291.698,A -85,B 0,C 180,E1 -24330.879,E2 -24330.879} C_VEL
LIN {X 0,Y 192.391,Z 293.442,A -85,B 0,C 180,E1 -24332.853,E2 -24332.853} C_VEL
LIN {X 0,Y 194.936,Z 297.112,A -85,B 0,C 180,E1 -24335.715,E2 -24335.715} C_VEL
LIN {X 0,Y 198.794,Z 302.692,A -85,B 0,C 180,E1 -24339.422,E2 -24339.422} C_VEL
LIN {X 0,Y 202.273,Z 307.847,A -85,B 0,C 180,E1 -24342.271,E2 -24342.271} C_VEL
LIN {X 0,Y 206.816,Z 314.796,A -85,B 0,C 180,E1 -24345.532,E2 -24345.532} C_VEL
LIN {X 0,Y 212.509,Z 324.281,A -85,B 0,C 180,E1 -24349.142,E2 -24349.142} C_VEL
LIN {X 0,Y 218.703,Z 335.355,A -85,B 0,C 180,E1 -24352.59,E2 -24352.59} C_VEL
LIN {X 0,Y 222.342,Z 342.397,A -85,B 0,C 180,E1 -24354.447,E2 -24354.447} C_VEL
LIN {X 0,Y 214.664,Z 424.306,A -85,B 0,C 180,E1 -24356.68,E2 -24356.68} C_VEL
LIN {X 0,Y 211.898,Z 441.307,A -85,B 0,C 180,E1 -24357.394,E2 -24357.394} C_VEL
LIN {X 0,Y 208.415,Z 457.12,A -85,B 0,C 180,E1 -24358.353,E2 -24358.353} C_VEL
LIN {X 0,Y 203.971,Z 473.063,A -85,B 0,C 180,E1 -24359.634,E2 -24359.634} C_VEL
LIN {X 0,Y 198.846,Z 488.277,A -85,B 0,C 180,E1 -24361.219,E2 -24361.219} C_VEL
LIN {X 0,Y 193.439,Z 501.94,A -85,B 0,C 180,E1 -24362.997,E2 -24362.997} C_VEL
LIN {X 0,Y 187.048,Z 515.914,A -85,B 0,C 180,E1 -24365.298,E2 -24365.298} C_VEL
LIN {X 0,Y 180.972,Z 527.817,A -85,B 0,C 180,E1 -24367.757,E2 -24367.757} C_VEL
LIN {X 0,Y 174.657,Z 539.102,A -85,B 0,C 180,E1 -24370.618,E2 -24370.618} C_VEL
LIN {X 0,Y 167.47,Z 551.069,A -85,B 0,C 180,E1 -24374.497,E2 -24374.497} C_VEL
LIN {X 0,Y 160.933,Z 561.132,A -85,B 0,C 180,E1 -24378.673,E2 -24378.673} C_VEL
LIN {X 0,Y 154.899,Z 570.155,A -85,B 0,C 180,E1 -24383.493,E2 -24383.493} C_VEL
LIN {X 0,Y 149.888,Z 577.663,A -85,B 0,C 180,E1 -24388.663,E2 -24388.663} C_VEL
LIN {X 0,Y 145.936,Z 583.852,A -85,B 0,C 180,E1 -24394.149,E2 -24394.149} C_VEL
LIN {X 0,Y 142.902,Z 589.133,A -85,B 0,C 180,E1 -24400.379,E2 -24400.379} C_VEL
LIN {X 0,Y 141.505,Z 591.729,A -85,B 0,C 180,E1 -24404.385,E2 -24404.385} C_VEL
LIN {X 0,Y 140.273,Z 594.622,A -85,B 0,C 180,E1 -24410.538,E2 -24410.538} C_VEL
LIN {X 0,Y 139.899,Z 596.426,A -85,B 0,C 180,E1 -24416.887,E2 -24416.887} C_VEL
LIN {X 0,Y 140.167,Z 597.01,A -85,B 0,C 180,E1 -24421.525,E2 -24421.525} C_VEL
LIN {X 0,Y 141.061,Z 596.957,A -85,B 0,C 180,E1 -24427.138,E2 -24427.138} C_VEL
LIN {X 0,Y 143.109,Z 595.733,A -85,B 0,C 180,E1 -24433.442,E2 -24433.442} C_VEL
LIN {X 0,Y 146.742,Z 593.149,A -85,B 0,C 180,E1 -24440.03,E2 -24440.03} C_VEL
LIN {X 0,Y 151.945,Z 589.133,A -85,B 0,C 180,E1 -24446.371,E2 -24446.371} C_VEL
LIN {X 0,Y 158.783,Z 583.585,A -85,B 0,C 180,E1 -24452.289,E2 -24452.289} C_VEL
LIN {X 0,Y 164.938,Z 578.311,A -85,B 0,C 180,E1 -24456.373,E2 -24456.373} C_VEL
LIN {X 0,Y 171.81,Z 572.028,A -85,B 0,C 180,E1 -24460.202,E2 -24460.202} C_VEL
LIN {X 0,Y 180.52,Z 563.487,A -85,B 0,C 180,E1 -24464.184,E2 -24464.184} C_VEL
LIN {X 0,Y 189.026,Z 554.309,A -85,B 0,C 180,E1 -24467.424,E2 -24467.424} C_VEL
LIN {X 0,Y 198.178,Z 543.405,A -85,B 0,C 180,E1 -24470.425,E2 -24470.425} C_VEL
LIN {X 0,Y 207.147,Z 531.548,A -85,B 0,C 180,E1 -24472.943,E2 -24472.943} C_VEL
LIN {X 0,Y 215.763,Z 518.613,A -85,B 0,C 180,E1 -24475.109,E2 -24475.109} C_VEL
LIN {X 0,Y 223.84,Z 504.639,A -85,B 0,C 180,E1 -24476.929,E2 -24476.929} C_VEL
LIN {X 0,Y 230.327,Z 491.609,A -85,B 0,C 180,E1 -24478.251,E2 -24478.251} C_VEL
LIN {X 0,Y 237.21,Z 475.37,A -85,B 0,C 180,E1 -24479.556,E2 -24479.556} C_VEL
LIN {X 0,Y 242.48,Z 460.07,A -85,B 0,C 180,E1 -24480.517,E2 -24480.517} C_VEL
LIN {X 0,Y 247.039,Z 443.199,A -85,B 0,C 180,E1 -24481.298,E2 -24481.298} C_VEL
LIN {X 0,Y 250.341,Z 426.408,A -85,B 0,C 180,E1 -24481.831,E2 -24481.831} C_VEL
LIN {X 0,Y 255.562,Z 382.732,A -85,B 0,C 180,E1 -24482.846,E2 -24482.846} C_VEL
LIN {X 0,Y 257.867,Z 362.58,A -85,B 0,C 180,E1 -24483.331,E2 -24483.331} C_VEL
LIN {X 0,Y 255.971,Z 357.413,A -85,B 0,C 180,E1 -24486.411,E2 -24486.411} C_VEL
LIN {X 0,Y 254.993,Z 355.02,A -85,B 0,C 180,E1 -24488.726,E2 -24488.726} C_VEL
LIN {X 0,Y 254.155,Z 353.577,A -85,B 0,C 180,E1 -24492.78,E2 -24492.78} C_VEL
LIN {X 0,Y 254.491,Z 354.634,A -85,B 0,C 180,E1 -24496.524,E2 -24496.524} C_VEL
LIN {X 0,Y 254.966,Z 355.421,A -85,B 0,C 180,E1 -24497.952,E2 -24497.952} C_VEL
LIN {X 0,Y 256.177,Z 358.615,A -85,B 0,C 180,E1 -24500.712,E2 -24500.712} C_VEL
LIN {X 0,Y 257.444,Z 362.027,A -85,B 0,C 180,E1 -24502.786,E2 -24502.786} C_VEL
LIN {X 0,Y 257.833,Z 363.496,A -85,B 0,C 180,E1 -24503.378,E2 -24503.378} C_VEL
LIN {X 0,Y 249.951,Z 430.148,A -85,B 0,C 180,E1 -24504.929,E2 -24504.929} C_VEL
LIN {X 0,Y 246.512,Z 447.461,A -85,B 0,C 180,E1 -24505.467,E2 -24505.467} C_VEL
LIN {X 0,Y 241.73,Z 464.471,A -85,B 0,C 180,E1 -24506.144,E2 -24506.144} C_VEL
LIN {X 0,Y 238.734,Z 473.355,A -85,B 0,C 180,E1 -24506.621,E2 -24506.621} C_VEL
LIN {X 0,Y 236.559,Z 478.819,A -85,B 0,C 180,E1 -24506.784,E2 -24506.784} C_VEL
LIN {X 0,Y 232.075,Z 487.683,A -85,B 0,C 180,E1 -24506.685,E2 -24506.685} C_VEL
LIN {X 0,Y 227.212,Z 496.284,A -85,B 0,C 180,E1 -24506.668,E2 -24506.668} C_VEL
LIN {X 0,Y 224.449,Z 501.327,A -85,B 0,C 180,E1 -24506.974,E2 -24506.974} C_VEL
LIN {X 0,Y 216.746,Z 515.226,A -85,B 0,C 180,E1 -24508.409,E2 -24508.409} C_VEL
LIN {X 0,Y 207.597,Z 529.452,A -85,B 0,C 180,E1 -24510.308,E2 -24510.308} C_VEL
LIN {X 0,Y 198.118,Z 542.4,A -85,B 0,C 180,E1 -24512.589,E2 -24512.589} C_VEL
LIN {X 0,Y 189.06,Z 553.449,A -85,B 0,C 180,E1 -24515.128,E2 -24515.128} C_VEL
LIN {X 0,Y 180.368,Z 563.035,A -85,B 0,C 180,E1 -24517.898,E2 -24517.898} C_VEL
LIN {X 0,Y 171.37,Z 572.105,A -85,B 0,C 180,E1 -24521.344,E2 -24521.344} C_VEL
LIN {X 0,Y 163.642,Z 579.335,A -85,B 0,C 180,E1 -24524.87,E2 -24524.87} C_VEL
LIN {X 0,Y 155.905,Z 586.107,A -85,B 0,C 180,E1 -24529.177,E2 -24529.177} C_VEL
LIN {X 0,Y 149.187,Z 591.705,A -85,B 0,C 180,E1 -24533.918,E2 -24533.918} C_VEL
LIN {X 0,Y 143.629,Z 596.287,A -85,B 0,C 180,E1 -24539.077,E2 -24539.077} C_VEL
LIN {X 0,Y 140.226,Z 599.042,A -85,B 0,C 180,E1 -24543.181,E2 -24543.181} C_VEL
LIN {X 0,Y 136.775,Z 601.804,A -85,B 0,C 180,E1 -24548.912,E2 -24548.912} C_VEL
LIN {X 0,Y 134.469,Z 603.717,A -85,B 0,C 180,E1 -24554.845,E2 -24554.845} C_VEL
LIN {X 0,Y 133.473,Z 604.603,A -85,B 0,C 180,E1 -24560.904,E2 -24560.904} C_VEL
LIN {X 0,Y 133.397,Z 604.632,A -85,B 0,C 180,E1 -24566.973,E2 -24566.973} C_VEL
LIN {X 0,Y 133.529,Z 604.228,A -85,B 0,C 180,E1 -24569.993,E2 -24569.993} C_VEL
LIN {X 0,Y 133.455,Z 603.589,A -85,B 0,C 180,E1 -24573.011,E2 -24573.011} C_VEL
LIN {X 0,Y 133.502,Z 601.581,A -85,B 0,C 180,E1 -24579.079,E2 -24579.079} C_VEL
LIN {X 0,Y 134.439,Z 598.419,A -85,B 0,C 180,E1 -24585.144,E2 -24585.144} C_VEL
LIN {X 0,Y 136.623,Z 594.229,A -85,B 0,C 180,E1 -24591.097,E2 -24591.097} C_VEL
LIN {X 0,Y 139.808,Z 588.78,A -85,B 0,C 180,E1 -24596.89,E2 -24596.89} C_VEL
LIN {X 0,Y 144.247,Z 582.059,A -85,B 0,C 180,E1 -24602.398,E2 -24602.398} C_VEL
LIN {X 0,Y 149.819,Z 573.939,A -85,B 0,C 180,E1 -24607.567,E2 -24607.567} C_VEL
LIN {X 0,Y 156.553,Z 564.209,A -85,B 0,C 180,E1 -24612.318,E2 -24612.318} C_VEL
LIN {X 0,Y 163.163,Z 554.052,A -85,B 0,C 180,E1 -24616.166,E2 -24616.166} C_VEL
LIN {X 0,Y 170.459,Z 542.145,A -85,B 0,C 180,E1 -24619.696,E2 -24619.696} C_VEL
LIN {X 0,Y 177.292,Z 530.24,A -85,B 0,C 180,E1 -24622.438,E2 -24622.438} C_VEL
LIN {X 0,Y 183.498,Z 518.084,A -85,B 0,C 180,E1 -24624.718,E2 -24624.718} C_VEL
LIN {X 0,Y 190.011,Z 503.798,A -85,B 0,C 180,E1 -24626.795,E2 -24626.795} C_VEL
LIN {X 0,Y 195.738,Z 489.063,A -85,B 0,C 180,E1 -24628.498,E2 -24628.498} C_VEL
LIN {X 0,Y 201.003,Z 473.087,A -85,B 0,C 180,E1 -24629.912,E2 -24629.912} C_VEL
LIN {X 0,Y 205.382,Z 456.641,A -85,B 0,C 180,E1 -24630.999,E2 -24630.999} C_VEL
LIN {X 0,Y 208.706,Z 440.563,A -85,B 0,C 180,E1 -24631.756,E2 -24631.756} C_VEL
LIN {X 0,Y 210.992,Z 423.355,A -85,B 0,C 180,E1 -24632.341,E2 -24632.341} C_VEL
LIN {X 0,Y 218.02,Z 348.138,A -85,B 0,C 180,E1 -24634.381,E2 -24634.381} C_VEL
LIN {X 0,Y 213.215,Z 336.739,A -85,B 0,C 180,E1 -24637.182,E2 -24637.182} C_VEL
LIN {X 0,Y 210.599,Z 331.454,A -85,B 0,C 180,E1 -24638.76,E2 -24638.76} C_VEL
LIN {X 0,Y 205.173,Z 321.984,A -85,B 0,C 180,E1 -24642.303,E2 -24642.303} C_VEL
LIN {X 0,Y 201.024,Z 315.266,A -85,B 0,C 180,E1 -24645.358,E2 -24645.358} C_VEL
LIN {X 0,Y 196.364,Z 307.858,A -85,B 0,C 180,E1 -24649.361,E2 -24649.361} C_VEL
LIN {X 0,Y 193.196,Z 303.277,A -85,B 0,C 180,E1 -24652.578,E2 -24652.578} C_VEL
LIN {X 0,Y 190.409,Z 298.986,A -85,B 0,C 180,E1 -24655.979,E2 -24655.979} C_VEL
LIN {X 0,Y 188.019,Z 295.588,A -85,B 0,C 180,E1 -24659.544,E2 -24659.544} C_VEL
LIN {X 0,Y 187.523,Z 294.474,A -85,B 0,C 180,E1 -24660.505,E2 -24660.505} C_VEL
LIN {X 0,Y 184.674,Z 290.542,A -85,B 0,C 180,E1 -24667.784,E2 -24667.784} C_VEL
LIN {X 0,Y 184.516,Z 289.808,A -85,B 0,C 180,E1 -24668.765,E2 -24668.765} C_VEL
LIN {X 0,Y 184.361,Z 290.004,A -85,B 0,C 180,E1 -24678.241,E2 -24678.241} C_VEL
LIN {X 0,Y 186.001,Z 293.755,A -85,B 0,C 180,E1 -24684.209,E2 -24684.209} C_VEL
LIN {X 0,Y 187.58,Z 295.223,A -85,B 0,C 180,E1 -24687.272,E2 -24687.272} C_VEL
LIN {X 0,Y 189.747,Z 298.788,A -85,B 0,C 180,E1 -24690.757,E2 -24690.757} C_VEL
LIN {X 0,Y 190.943,Z 300.236,A -85,B 0,C 180,E1 -24692.337,E2 -24692.337} C_VEL
LIN {X 0,Y 193.53,Z 303.937,A -85,B 0,C 180,E1 -24695.343,E2 -24695.343} C_VEL
LIN {X 0,Y 197.212,Z 309.577,A -85,B 0,C 180,E1 -24698.999,E2 -24698.999} C_VEL
LIN {X 0,Y 200.661,Z 314.832,A -85,B 0,C 180,E1 -24701.895,E2 -24701.895} C_VEL
LIN {X 0,Y 205.416,Z 322.422,A -85,B 0,C 180,E1 -24705.402,E2 -24705.402} C_VEL
LIN {X 0,Y 210.332,Z 331.028,A -85,B 0,C 180,E1 -24708.608,E2 -24708.608} C_VEL
LIN {X 0,Y 215.61,Z 340.649,A -85,B 0,C 180,E1 -24711.653,E2 -24711.653} C_VEL
LIN {X 0,Y 218.034,Z 345.506,A -85,B 0,C 180,E1 -24712.975,E2 -24712.975} C_VEL
LIN {X 0,Y 210.489,Z 424.202,A -85,B 0,C 180,E1 -24715.132,E2 -24715.132} C_VEL
LIN {X 0,Y 207.497,Z 442.157,A -85,B 0,C 180,E1 -24715.884,E2 -24715.884} C_VEL
LIN {X 0,Y 203.592,Z 459.088,A -85,B 0,C 180,E1 -24716.925,E2 -24716.925} C_VEL
LIN {X 0,Y 199.411,Z 473.424,A -85,B 0,C 180,E1 -24718.092,E2 -24718.092} C_VEL
LIN {X 0,Y 193.766,Z 489.571,A -85,B 0,C 180,E1 -24719.792,E2 -24719.792} C_VEL
LIN {X 0,Y 187.612,Z 504.374,A -85,B 0,C 180,E1 -24721.782,E2 -24721.782} C_VEL
LIN {X 0,Y 181.035,Z 518.097,A -85,B 0,C 180,E1 -24724.111,E2 -24724.111} C_VEL
LIN {X 0,Y 174.249,Z 530.713,A -85,B 0,C 180,E1 -24726.85,E2 -24726.85} C_VEL
LIN {X 0,Y 167.8,Z 541.564,A -85,B 0,C 180,E1 -24729.792,E2 -24729.792} C_VEL
LIN {X 0,Y 160.742,Z 552.725,A -85,B 0,C 180,E1 -24733.625,E2 -24733.625} C_VEL
LIN {X 0,Y 154.598,Z 561.793,A -85,B 0,C 180,E1 -24737.537,E2 -24737.537} C_VEL
LIN {X 0,Y 148.298,Z 570.744,A -85,B 0,C 180,E1 -24742.519,E2 -24742.519} C_VEL
LIN {X 0,Y 143.648,Z 577.338,A -85,B 0,C 180,E1 -24747.203,E2 -24747.203} C_VEL
LIN {X 0,Y 139.424,Z 583.638,A -85,B 0,C 180,E1 -24752.896,E2 -24752.896} C_VEL
LIN {X 0,Y 136.304,Z 588.614,A -85,B 0,C 180,E1 -24758.905,E2 -24758.905} C_VEL
LIN {X 0,Y 134.149,Z 592.48,A -85,B 0,C 180,E1 -24765.192,E2 -24765.192} C_VEL
LIN {X 0,Y 133.473,Z 594.069,A -85,B 0,C 180,E1 -24768.591,E2 -24768.591} C_VEL
LIN {X 0,Y 132.849,Z 596.182,A -85,B 0,C 180,E1 -24775.045,E2 -24775.045} C_VEL
LIN {X 0,Y 133.099,Z 597.203,A -85,B 0,C 180,E1 -24781.88,E2 -24781.88} C_VEL
LIN {X 0,Y 134.355,Z 597.058,A -85,B 0,C 180,E1 -24788.889,E2 -24788.889} C_VEL
LIN {X 0,Y 137.061,Z 595.641,A -85,B 0,C 180,E1 -24795.887,E2 -24795.887} C_VEL
LIN {X 0,Y 141.357,Z 592.803,A -85,B 0,C 180,E1 -24802.71,E2 -24802.71} C_VEL
LIN {X 0,Y 147.287,Z 588.514,A -85,B 0,C 180,E1 -24809.202,E2 -24809.202} C_VEL
LIN {X 0,Y 154.918,Z 582.677,A -85,B 0,C 180,E1 -24815.148,E2 -24815.148} C_VEL
LIN {X 0,Y 162.643,Z 576.379,A -85,B 0,C 180,E1 -24819.775,E2 -24819.775} C_VEL
LIN {X 0,Y 171.699,Z 568.347,A -85,B 0,C 180,E1 -24824.142,E2 -24824.142} C_VEL
LIN {X 0,Y 180,Z 560.197,A -85,B 0,C 180,E1 -24827.466,E2 -24827.466} C_VEL
LIN {X 0,Y 188.851,Z 550.763,A -85,B 0,C 180,E1 -24830.483,E2 -24830.483} C_VEL
LIN {X 0,Y 198.178,Z 539.735,A -85,B 0,C 180,E1 -24833.222,E2 -24833.222} C_VEL
LIN {X 0,Y 207.804,Z 526.828,A -85,B 0,C 180,E1 -24835.668,E2 -24835.668} C_VEL
LIN {X 0,Y 216.312,Z 513.73,A -85,B 0,C 180,E1 -24837.583,E2 -24837.583} C_VEL
LIN {X 0,Y 223.195,Z 501.679,A -85,B 0,C 180,E1 -24838.991,E2 -24838.991} C_VEL
LIN {X 0,Y 229.478,Z 489.113,A -85,B 0,C 180,E1 -24840.19,E2 -24840.19} C_VEL
LIN {X 0,Y 236.027,Z 473.504,A -85,B 0,C 180,E1 -24841.358,E2 -24841.358} C_VEL
LIN {X 0,Y 240.892,Z 459.341,A -85,B 0,C 180,E1 -24842.188,E2 -24842.188} C_VEL
LIN {X 0,Y 245.313,Z 443.17,A -85,B 0,C 180,E1 -24842.901,E2 -24842.901} C_VEL
LIN {X 0,Y 248.644,Z 426.593,A -85,B 0,C 180,E1 -24843.408,E2 -24843.408} C_VEL
LIN {X 0,Y 253.416,Z 388.069,A -85,B 0,C 180,E1 -24844.293,E2 -24844.293} C_VEL
LIN {X 0,Y 255.86,Z 367.411,A -85,B 0,C 180,E1 -24844.781,E2 -24844.781} C_VEL
LIN {X 0,Y 254.544,Z 363.685,A -85,B 0,C 180,E1 -24847.295,E2 -24847.295} C_VEL
LIN {X 0,Y 254.014,Z 362.044,A -85,B 0,C 180,E1 -24848.76,E2 -24848.76} C_VEL
LIN {X 0,Y 253.193,Z 360.597,A -85,B 0,C 180,E1 -24852.829,E2 -24852.829} C_VEL
LIN {X 0,Y 253.701,Z 361.903,A -85,B 0,C 180,E1 -24857.073,E2 -24857.073} C_VEL
LIN {X 0,Y 254.77,Z 364.837,A -85,B 0,C 180,E1 -24859.956,E2 -24859.956} C_VEL
LIN {X 0,Y 255.86,Z 367.895,A -85,B 0,C 180,E1 -24861.918,E2 -24861.918} C_VEL
LIN {X 0,Y 248.343,Z 429.479,A -85,B 0,C 180,E1 -24863.323,E2 -24863.323} C_VEL
LIN {X 0,Y 244.87,Z 446.762,A -85,B 0,C 180,E1 -24863.841,E2 -24863.841} C_VEL
LIN {X 0,Y 240.533,Z 462.239,A -85,B 0,C 180,E1 -24864.428,E2 -24864.428} C_VEL
LIN {X 0,Y 235.019,Z 477.867,A -85,B 0,C 180,E1 -24865.227,E2 -24865.227} C_VEL
LIN {X 0,Y 229.054,Z 491.919,A -85,B 0,C 180,E1 -24866.168,E2 -24866.168} C_VEL
LIN {X 0,Y 224.449,Z 501.327,A -85,B 0,C 180,E1 -24866.974,E2 -24866.974} C_VEL
LIN {X 0,Y 221.566,Z 506.444,A -85,B 0,C 180,E1 -24867.316,E2 -24867.316} C_VEL
LIN {X 0,Y 211.227,Z 520.917,A -85,B 0,C 180,E1 -24867.579,E2 -24867.579} C_VEL
LIN {X 0,Y 207.802,Z 525.535,A -85,B 0,C 180,E1 -24867.905,E2 -24867.905} C_VEL
LIN {X 0,Y 206.744,Z 527.009,A -85,B 0,C 180,E1 -24868.09,E2 -24868.09} C_VEL
LIN {X 0,Y 197.323,Z 539.752,A -85,B 0,C 180,E1 -24870.156,E2 -24870.156} C_VEL
LIN {X 0,Y 187.732,Z 551.331,A -85,B 0,C 180,E1 -24872.608,E2 -24872.608} C_VEL
LIN {X 0,Y 177.371,Z 562.422,A -85,B 0,C 180,E1 -24875.675,E2 -24875.675} C_VEL
LIN {X 0,Y 167.841,Z 571.567,A -85,B 0,C 180,E1 -24879.057,E2 -24879.057} C_VEL
LIN {X 0,Y 158.687,Z 579.689,A -85,B 0,C 180,E1 -24883.043,E2 -24883.043} C_VEL
LIN {X 0,Y 150.573,Z 586.401,A -85,B 0,C 180,E1 -24887.4,E2 -24887.4} C_VEL
LIN {X 0,Y 143.438,Z 591.869,A -85,B 0,C 180,E1 -24892.226,E2 -24892.226} C_VEL
LIN {X 0,Y 136.195,Z 597.285,A -85,B 0,C 180,E1 -24898.927,E2 -24898.927} C_VEL
LIN {X 0,Y 131.439,Z 600.825,A -85,B 0,C 180,E1 -24905.362,E2 -24905.362} C_VEL
LIN {X 0,Y 127.559,Z 603.582,A -85,B 0,C 180,E1 -24914.002,E2 -24914.002} C_VEL
LIN {X 0,Y 126.406,Z 604.415,A -85,B 0,C 180,E1 -24920.391,E2 -24920.391} C_VEL
LIN {X 0,Y 126.295,Z 604.39,A -85,B 0,C 180,E1 -24926.802,E2 -24926.802} C_VEL
LIN {X 0,Y 126.442,Z 603.959,A -85,B 0,C 180,E1 -24929.992,E2 -24929.992} C_VEL
LIN {X 0,Y 126.364,Z 603.278,A -85,B 0,C 180,E1 -24933.18,E2 -24933.18} C_VEL
LIN {X 0,Y 126.457,Z 601.2,A -85,B 0,C 180,E1 -24939.59,E2 -24939.59} C_VEL
LIN {X 0,Y 128.048,Z 597.052,A -85,B 0,C 180,E1 -24947.561,E2 -24947.561} C_VEL
LIN {X 0,Y 131.476,Z 591.114,A -85,B 0,C 180,E1 -24955.308,E2 -24955.308} C_VEL
LIN {X 0,Y 135.611,Z 584.933,A -85,B 0,C 180,E1 -24961.205,E2 -24961.205} C_VEL
LIN {X 0,Y 141.02,Z 577.428,A -85,B 0,C 180,E1 -24966.72,E2 -24966.72} C_VEL
LIN {X 0,Y 147.583,Z 568.414,A -85,B 0,C 180,E1 -24971.801,E2 -24971.801} C_VEL
LIN {X 0,Y 155.146,Z 557.61,A -85,B 0,C 180,E1 -24976.44,E2 -24976.44} C_VEL
LIN {X 0,Y 162.502,Z 546.401,A -85,B 0,C 180,E1 -24980.133,E2 -24980.133} C_VEL
LIN {X 0,Y 169.317,Z 535.122,A -85,B 0,C 180,E1 -24983.025,E2 -24983.025} C_VEL
LIN {X 0,Y 175.96,Z 523.221,A -85,B 0,C 180,E1 -24985.452,E2 -24985.452} C_VEL
LIN {X 0,Y 182.867,Z 509.265,A -85,B 0,C 180,E1 -24987.713,E2 -24987.713} C_VEL
LIN {X 0,Y 188.105,Z 497.248,A -85,B 0,C 180,E1 -24989.227,E2 -24989.227} C_VEL
LIN {X 0,Y 193.393,Z 483.15,A -85,B 0,C 180,E1 -24990.698,E2 -24990.698} C_VEL
LIN {X 0,Y 198.521,Z 466.959,A -85,B 0,C 180,E1 -24991.971,E2 -24991.971} C_VEL
LIN {X 0,Y 202.537,Z 450.953,A -85,B 0,C 180,E1 -24992.892,E2 -24992.892} C_VEL
LIN {X 0,Y 205.636,Z 434.055,A -85,B 0,C 180,E1 -24993.585,E2 -24993.585} C_VEL
LIN {X 0,Y 208.308,Z 409.254,A -85,B 0,C 180,E1 -24994.326,E2 -24994.326} C_VEL
LIN {X 0,Y 213.956,Z 351.093,A -85,B 0,C 180,E1 -24995.868,E2 -24995.868} C_VEL
LIN {X 0,Y 209.771,Z 341.097,A -85,B 0,C 180,E1 -24998.44,E2 -24998.44} C_VEL
LIN {X 0,Y 207.698,Z 336.829,A -85,B 0,C 180,E1 -24999.772,E2 -24999.772} C_VEL
LIN {X 0,Y 202.548,Z 327.628,A -85,B 0,C 180,E1 -25003.302,E2 -25003.302} C_VEL
LIN {X 0,Y 198.942,Z 321.507,A -85,B 0,C 180,E1 -25006.123,E2 -25006.123} C_VEL
LIN {X 0,Y 194.512,Z 314.264,A -85,B 0,C 180,E1 -25010.097,E2 -25010.097} C_VEL
LIN {X 0,Y 191.703,Z 310.009,A -85,B 0,C 180,E1 -25013.065,E2 -25013.065} C_VEL
LIN {X 0,Y 188.932,Z 305.707,A -85,B 0,C 180,E1 -25016.601,E2 -25016.601} C_VEL
LIN {X 0,Y 186.502,Z 301.841,A -85,B 0,C 180,E1 -25020.508,E2 -25020.508} C_VEL
LIN {X 0,Y 185.773,Z 300.842,A -85,B 0,C 180,E1 -25021.954,E2 -25021.954} C_VEL
LIN {X 0,Y 183.577,Z 297.224,A -85,B 0,C 180,E1 -25028.498,E2 -25028.498} C_VEL
LIN {X 0,Y 183.358,Z 296.77,A -85,B 0,C 180,E1 -25029.67,E2 -25029.67} C_VEL
LIN {X 0,Y 183.333,Z 296.951,A -85,B 0,C 180,E1 -25037.86,E2 -25037.86} C_VEL
LIN {X 0,Y 184.938,Z 300.716,A -85,B 0,C 180,E1 -25044.004,E2 -25044.004} C_VEL
LIN {X 0,Y 186.31,Z 302.055,A -85,B 0,C 180,E1 -25046.766,E2 -25046.766} C_VEL
LIN {X 0,Y 188.388,Z 305.566,A -85,B 0,C 180,E1 -25050.266,E2 -25050.266} C_VEL
LIN {X 0,Y 189.506,Z 306.995,A -85,B 0,C 180,E1 -25051.802,E2 -25051.802} C_VEL
LIN {X 0,Y 192.699,Z 311.886,A -85,B 0,C 180,E1 -25055.61,E2 -25055.61} C_VEL
LIN {X 0,Y 195.4,Z 316.079,A -85,B 0,C 180,E1 -25058.343,E2 -25058.343} C_VEL
LIN {X 0,Y 199.424,Z 322.351,A -85,B 0,C 180,E1 -25061.812,E2 -25061.812} C_VEL
LIN {X 0,Y 204.034,Z 330.261,A -85,B 0,C 180,E1 -25065.298,E2 -25065.298} C_VEL
LIN {X 0,Y 209.047,Z 339.272,A -85,B 0,C 180,E1 -25068.603,E2 -25068.603} C_VEL
LIN {X 0,Y 213.918,Z 348.736,A -85,B 0,C 180,E1 -25071.477,E2 -25071.477} C_VEL
LIN {X 0,Y 206.485,Z 424.057,A -85,B 0,C 180,E1 -25073.525,E2 -25073.525} C_VEL
LIN {X 0,Y 203.578,Z 441.221,A -85,B 0,C 180,E1 -25074.224,E2 -25074.224} C_VEL
LIN {X 0,Y 199.894,Z 457.174,A -85,B 0,C 180,E1 -25075.165,E2 -25075.165} C_VEL
LIN {X 0,Y 195.292,Z 472.962,A -85,B 0,C 180,E1 -25076.414,E2 -25076.414} C_VEL
LIN {X 0,Y 190.105,Z 487.617,A -85,B 0,C 180,E1 -25077.898,E2 -25077.898} C_VEL
LIN {X 0,Y 183.72,Z 502.839,A -85,B 0,C 180,E1 -25079.87,E2 -25079.87} C_VEL
LIN {X 0,Y 176.902,Z 516.76,A -85,B 0,C 180,E1 -25082.18,E2 -25082.18} C_VEL
LIN {X 0,Y 169.7,Z 529.873,A -85,B 0,C 180,E1 -25084.983,E2 -25084.983} C_VEL
LIN {X 0,Y 162.031,Z 542.34,A -85,B 0,C 180,E1 -25088.373,E2 -25088.373} C_VEL
LIN {X 0,Y 155.193,Z 552.696,A -85,B 0,C 180,E1 -25091.994,E2 -25091.994} C_VEL
LIN {X 0,Y 148.312,Z 562.424,A -85,B 0,C 180,E1 -25096.302,E2 -25096.302} C_VEL
LIN {X 0,Y 141.752,Z 571.311,A -85,B 0,C 180,E1 -25101.453,E2 -25101.453} C_VEL
LIN {X 0,Y 136.294,Z 578.677,A -85,B 0,C 180,E1 -25107.051,E2 -25107.051} C_VEL
LIN {X 0,Y 131.987,Z 584.735,A -85,B 0,C 180,E1 -25113.06,E2 -25113.06} C_VEL
LIN {X 0,Y 128.921,Z 589.587,A -85,B 0,C 180,E1 -25119.42,E2 -25119.42} C_VEL
LIN {X 0,Y 126.801,Z 593.225,A -85,B 0,C 180,E1 -25126.096,E2 -25126.096} C_VEL
LIN {X 0,Y 125.804,Z 595.786,A -85,B 0,C 180,E1 -25133.028,E2 -25133.028} C_VEL
LIN {X 0,Y 125.731,Z 596.661,A -85,B 0,C 180,E1 -25136.57,E2 -25136.57} C_VEL
LIN {X 0,Y 126.199,Z 597.499,A -85,B 0,C 180,E1 -25143.849,E2 -25143.849} C_VEL
LIN {X 0,Y 127.916,Z 597.106,A -85,B 0,C 180,E1 -25151.255,E2 -25151.255} C_VEL
LIN {X 0,Y 131.218,Z 595.443,A -85,B 0,C 180,E1 -25158.585,E2 -25158.585} C_VEL
LIN {X 0,Y 136.27,Z 592.42,A -85,B 0,C 180,E1 -25165.617,E2 -25165.617} C_VEL
LIN {X 0,Y 143.042,Z 587.912,A -85,B 0,C 180,E1 -25172.186,E2 -25172.186} C_VEL
LIN {X 0,Y 151.476,Z 581.821,A -85,B 0,C 180,E1 -25178.127,E2 -25178.127} C_VEL
LIN {X 0,Y 159.537,Z 575.466,A -85,B 0,C 180,E1 -25182.558,E2 -25182.558} C_VEL
LIN {X 0,Y 169.539,Z 566.892,A -85,B 0,C 180,E1 -25186.961,E2 -25186.961} C_VEL
LIN {X 0,Y 178.332,Z 558.622,A -85,B 0,C 180,E1 -25190.163,E2 -25190.163} C_VEL
LIN {X 0,Y 188.819,Z 547.521,A -85,B 0,C 180,E1 -25193.417,E2 -25193.417} C_VEL
LIN {X 0,Y 199.105,Z 535.231,A -85,B 0,C 180,E1 -25196.104,E2 -25196.104} C_VEL
LIN {X 0,Y 207.573,Z 523.753,A -85,B 0,C 180,E1 -25198.059,E2 -25198.059} C_VEL
LIN {X 0,Y 216.017,Z 510.763,A -85,B 0,C 180,E1 -25199.813,E2 -25199.813} C_VEL
LIN {X 0,Y 224.085,Z 496.365,A -85,B 0,C 180,E1 -25201.323,E2 -25201.323} C_VEL
LIN {X 0,Y 231.376,Z 480.893,A -85,B 0,C 180,E1 -25202.556,E2 -25202.556} C_VEL
LIN {X 0,Y 237.188,Z 465.817,A -85,B 0,C 180,E1 -25203.525,E2 -25203.525} C_VEL
LIN {X 0,Y 242.278,Z 449.334,A -85,B 0,C 180,E1 -25204.304,E2 -25204.304} C_VEL
LIN {X 0,Y 245.989,Z 433.395,A -85,B 0,C 180,E1 -25204.849,E2 -25204.849} C_VEL
LIN {X 0,Y 248.749,Z 415.781,A -85,B 0,C 180,E1 -25205.286,E2 -25205.286} C_VEL
LIN {X 0,Y 254.018,Z 372.529,A -85,B 0,C 180,E1 -25206.225,E2 -25206.225} C_VEL
LIN {X 0,Y 253.284,Z 370.156,A -85,B 0,C 180,E1 -25207.974,E2 -25207.974} C_VEL
LIN {X 0,Y 252.856,Z 368.889,A -85,B 0,C 180,E1 -25209.263,E2 -25209.263} C_VEL
LIN {X 0,Y 252.227,Z 367.645,A -85,B 0,C 180,E1 -25212.879,E2 -25212.879} C_VEL
LIN {X 0,Y 252.757,Z 368.985,A -85,B 0,C 180,E1 -25217.138,E2 -25217.138} C_VEL
LIN {X 0,Y 253.856,Z 372.515,A -85,B 0,C 180,E1 -25220.163,E2 -25220.163} C_VEL
LIN {X 0,Y 254,Z 372.899,A -85,B 0,C 180,E1 -25220.437,E2 -25220.437} C_VEL
LIN {X 0,Y 246.883,Z 429.701,A -85,B 0,C 180,E1 -25221.719,E2 -25221.719} C_VEL
LIN {X 0,Y 243.16,Z 447.569,A -85,B 0,C 180,E1 -25222.239,E2 -25222.239} C_VEL
LIN {X 0,Y 238.744,Z 462.714,A -85,B 0,C 180,E1 -25222.793,E2 -25222.793} C_VEL
LIN {X 0,Y 233.69,Z 476.72,A -85,B 0,C 180,E1 -25223.466,E2 -25223.466} C_VEL
LIN {X 0,Y 226.839,Z 492.432,A -85,B 0,C 180,E1 -25224.475,E2 -25224.475} C_VEL
LIN {X 0,Y 219.428,Z 506.807,A -85,B 0,C 180,E1 -25225.73,E2 -25225.73} C_VEL
LIN {X 0,Y 211.357,Z 520.135,A -85,B 0,C 180,E1 -25227.186,E2 -25227.186} C_VEL
LIN {X 0,Y 206.744,Z 527.009,A -85,B 0,C 180,E1 -25228.09,E2 -25228.09} C_VEL
LIN {X 0,Y 203.306,Z 531.561,A -85,B 0,C 180,E1 -25228.573,E2 -25228.573} C_VEL
LIN {X 0,Y 190.598,Z 545.162,A -85,B 0,C 180,E1 -25229.429,E2 -25229.429} C_VEL
LIN {X 0,Y 187.41,Z 548.462,A -85,B 0,C 180,E1 -25229.915,E2 -25229.915} C_VEL
LIN {X 0,Y 186.248,Z 549.75,A -85,B 0,C 180,E1 -25230.184,E2 -25230.184} C_VEL
LIN {X 0,Y 175.961,Z 560.477,A -85,B 0,C 180,E1 -25232.985,E2 -25232.985} C_VEL
LIN {X 0,Y 165.688,Z 570.11,A -85,B 0,C 180,E1 -25236.294,E2 -25236.294} C_VEL
LIN {X 0,Y 156.172,Z 578.293,A -85,B 0,C 180,E1 -25240.083,E2 -25240.083} C_VEL
LIN {X 0,Y 145.381,Z 586.66,A -85,B 0,C 180,E1 -25245.489,E2 -25245.489} C_VEL
LIN {X 0,Y 136.156,Z 593.282,A -85,B 0,C 180,E1 -25251.72,E2 -25251.72} C_VEL
LIN {X 0,Y 130.092,Z 597.348,A -85,B 0,C 180,E1 -25257.293,E2 -25257.293} C_VEL
LIN {X 0,Y 124.678,Z 600.933,A -85,B 0,C 180,E1 -25264.406,E2 -25264.406} C_VEL
LIN {X 0,Y 120.689,Z 603.441,A -85,B 0,C 180,E1 -25273.065,E2 -25273.065} C_VEL
LIN {X 0,Y 119.365,Z 604.229,A -85,B 0,C 180,E1 -25279.818,E2 -25279.818} C_VEL
LIN {X 0,Y 119.184,Z 604.12,A -85,B 0,C 180,E1 -25286.611,E2 -25286.611} C_VEL
LIN {X 0,Y 119.356,Z 603.691,A -85,B 0,C 180,E1 -25289.992,E2 -25289.992} C_VEL
LIN {X 0,Y 119.266,Z 602.966,A -85,B 0,C 180,E1 -25293.37,E2 -25293.37} C_VEL
LIN {X 0,Y 119.401,Z 600.799,A -85,B 0,C 180,E1 -25300.162,E2 -25300.162} C_VEL
LIN {X 0,Y 120.655,Z 597.526,A -85,B 0,C 180,E1 -25306.923,E2 -25306.923} C_VEL
LIN {X 0,Y 123.228,Z 593.138,A -85,B 0,C 180,E1 -25313.52,E2 -25313.52} C_VEL
LIN {X 0,Y 127.071,Z 587.59,A -85,B 0,C 180,E1 -25319.842,E2 -25319.842} C_VEL
LIN {X 0,Y 132.239,Z 580.657,A -85,B 0,C 180,E1 -25325.764,E2 -25325.764} C_VEL
LIN {X 0,Y 138.636,Z 572.307,A -85,B 0,C 180,E1 -25331.214,E2 -25331.214} C_VEL
LIN {X 0,Y 145.165,Z 563.704,A -85,B 0,C 180,E1 -25335.558,E2 -25335.558} C_VEL
LIN {X 0,Y 152.908,Z 552.73,A -85,B 0,C 180,E1 -25339.836,E2 -25339.836} C_VEL
LIN {X 0,Y 160.271,Z 541.589,A -85,B 0,C 180,E1 -25343.143,E2 -25343.143} C_VEL
LIN {X 0,Y 168.221,Z 528.552,A -85,B 0,C 180,E1 -25346.12,E2 -25346.12} C_VEL
LIN {X 0,Y 174.95,Z 515.969,A -85,B 0,C 180,E1 -25348.418,E2 -25348.418} C_VEL
LIN {X 0,Y 181.165,Z 503.135,A -85,B 0,C 180,E1 -25350.212,E2 -25350.212} C_VEL
LIN {X 0,Y 187.198,Z 488.309,A -85,B 0,C 180,E1 -25351.901,E2 -25351.901} C_VEL
LIN {X 0,Y 192.752,Z 472.237,A -85,B 0,C 180,E1 -25353.276,E2 -25353.276} C_VEL
LIN {X 0,Y 197.358,Z 455.647,A -85,B 0,C 180,E1 -25354.325,E2 -25354.325} C_VEL
LIN {X 0,Y 200.846,Z 439.114,A -85,B 0,C 180,E1 -25355.071,E2 -25355.071} C_VEL
LIN {X 0,Y 203.189,Z 422.124,A -85,B 0,C 180,E1 -25355.622,E2 -25355.622} C_VEL
LIN {X 0,Y 209.955,Z 353.949,A -85,B 0,C 180,E1 -25357.425,E2 -25357.425} C_VEL
LIN {X 0,Y 205.808,Z 343.96,A -85,B 0,C 180,E1 -25360.176,E2 -25360.176} C_VEL
LIN {X 0,Y 200.992,Z 335.032,A -85,B 0,C 180,E1 -25363.561,E2 -25363.561} C_VEL
LIN {X 0,Y 197.074,Z 328.052,A -85,B 0,C 180,E1 -25366.726,E2 -25366.726} C_VEL
LIN {X 0,Y 192.743,Z 320.726,A -85,B 0,C 180,E1 -25370.795,E2 -25370.795} C_VEL
LIN {X 0,Y 189.841,Z 316.277,A -85,B 0,C 180,E1 -25374,E2 -25374} C_VEL
LIN {X 0,Y 187.48,Z 312.371,A -85,B 0,C 180,E1 -25377.222,E2 -25377.222} C_VEL
LIN {X 0,Y 185.2,Z 308.551,A -85,B 0,C 180,E1 -25381.111,E2 -25381.111} C_VEL
LIN {X 0,Y 182.393,Z 303.793,A -85,B 0,C 180,E1 -25389.721,E2 -25389.721} C_VEL
LIN {X 0,Y 182.346,Z 304.01,A -85,B 0,C 180,E1 -25397.729,E2 -25397.729} C_VEL
LIN {X 0,Y 183.777,Z 307.61,A -85,B 0,C 180,E1 -25403.572,E2 -25403.572} C_VEL
LIN {X 0,Y 185.102,Z 309,A -85,B 0,C 180,E1 -25406.357,E2 -25406.357} C_VEL
LIN {X 0,Y 187.298,Z 312.624,A -85,B 0,C 180,E1 -25410.145,E2 -25410.145} C_VEL
LIN {X 0,Y 188.333,Z 314.276,A -85,B 0,C 180,E1 -25411.629,E2 -25411.629} C_VEL
LIN {X 0,Y 190.836,Z 318.133,A -85,B 0,C 180,E1 -25414.742,E2 -25414.742} C_VEL
LIN {X 0,Y 193.68,Z 322.695,A -85,B 0,C 180,E1 -25417.743,E2 -25417.743} C_VEL
LIN {X 0,Y 197.475,Z 328.831,A -85,B 0,C 180,E1 -25421.154,E2 -25421.154} C_VEL
LIN {X 0,Y 201.742,Z 336.454,A -85,B 0,C 180,E1 -25424.535,E2 -25424.535} C_VEL
LIN {X 0,Y 206.296,Z 344.887,A -85,B 0,C 180,E1 -25427.669,E2 -25427.669} C_VEL
LIN {X 0,Y 209.886,Z 352.067,A -85,B 0,C 180,E1 -25429.933,E2 -25429.933} C_VEL
LIN {X 0,Y 202.47,Z 424.85,A -85,B 0,C 180,E1 -25431.895,E2 -25431.895} C_VEL
LIN {X 0,Y 199.326,Z 442.721,A -85,B 0,C 180,E1 -25432.627,E2 -25432.627} C_VEL
LIN {X 0,Y 195.04,Z 460.264,A -85,B 0,C 180,E1 -25433.687,E2 -25433.687} C_VEL
LIN {X 0,Y 189.985,Z 476.407,A -85,B 0,C 180,E1 -25435.021,E2 -25435.021} C_VEL
LIN {X 0,Y 184.199,Z 491.592,A -85,B 0,C 180,E1 -25436.648,E2 -25436.648} C_VEL
LIN {X 0,Y 177.484,Z 506.517,A -85,B 0,C 180,E1 -25438.694,E2 -25438.694} C_VEL
LIN {X 0,Y 170.519,Z 519.948,A -85,B 0,C 180,E1 -25441.042,E2 -25441.042} C_VEL
LIN {X 0,Y 163.269,Z 532.449,A -85,B 0,C 180,E1 -25443.83,E2 -25443.83} C_VEL
LIN {X 0,Y 155.303,Z 544.768,A -85,B 0,C 180,E1 -25447.385,E2 -25447.385} C_VEL
LIN {X 0,Y 148.034,Z 555.075,A -85,B 0,C 180,E1 -25451.244,E2 -25451.244} C_VEL
LIN {X 0,Y 141.202,Z 564.186,A -85,B 0,C 180,E1 -25455.597,E2 -25455.597} C_VEL
